MoveL RelTool (p1,32.000000,16.000000,15.618348,\Rx:=0.000000,\Ry:=-3.162780),vel1,zoneval,Extruder\WObj:=Workobject_1;
MoveL RelTool (p1,34.500000,16.000000,16.195789,\Rx:=0.000000,\Ry:=-2.451727),vel1,zoneval,Extruder\WObj:=Workobject_1;
MoveL RelTool (p1,37.000000,16.000000,16.604171,\Rx:=0.000000,\Ry:=-1.580071),vel1,zoneval,Extruder\WObj:=Workobject_1;
MoveL RelTool (p1,39.500000,16.000000,16.864821,\Rx:=0.000000,\Ry:=-1.023091),vel1,zoneval,Extruder\WObj:=Workobject_1;
MoveL RelTool (p1,42.000000,16.000000,16.985827,\Rx:=0.000000,\Ry:=-0.098788),vel1,zoneval,Extruder\WObj:=Workobject_1;
MoveL RelTool (p1,44.500000,16.000000,16.964311,\Rx:=0.000000,\Ry:=0.392042),vel1,zoneval,Extruder\WObj:=Workobject_1;
MoveL RelTool (p1,47.000000,16.000000,16.814464,\Rx:=0.000000,\Ry:=1.375711),vel1,zoneval,Extruder\WObj:=Workobject_1;
MoveL RelTool (p1,49.500000,16.000000,16.508665,\Rx:=0.000000,\Ry:=1.876566),vel1,zoneval,Extruder\WObj:=Workobject_1;
MoveL RelTool (p1,52.000000,16.000000,16.062619,\Rx:=0.000000,\Ry:=2.914714),vel1,zoneval,Extruder\WObj:=Workobject_1;
MoveL RelTool (p1,54.500000,16.000000,15.430893,\Rx:=0.000000,\Ry:=3.587334),vel1,zoneval,Extruder\WObj:=Workobject_1;
MoveL RelTool (p1,57.000000,16.000000,14.596569,\Rx:=0.000000,\Ry:=4.605885),vel1,zoneval,Extruder\WObj:=Workobject_1;
MoveL RelTool (p1,59.500000,16.000000,13.508587,\Rx:=0.000000,\Ry:=5.885518),vel1,zoneval,Extruder\WObj:=Workobject_1;
MoveL RelTool (p1,62.000000,16.000000,12.049469,\Rx:=0.000000,\Ry:=8.052866),vel1,zoneval,Extruder\WObj:=Workobject_1;
MoveL RelTool (p1,64.500000,16.000000,9.870531,\Rx:=0.000000,\Ry:=11.251023),vel1,zoneval,Extruder\WObj:=Workobject_1;
MoveL RelTool (p1,67.000000,16.000000,7.452288,\Rx:=0.000000,\Ry:=5.136110),vel1,zoneval,Extruder\WObj:=Workobject_1;
MoveL RelTool (p1,69.500000,16.000000,7.000000,\Rx:=0.000000,\Ry:=-0.000000),vel1,zoneval,Extruder\WObj:=Workobject_1;
MoveL RelTool (p1,72.000000,16.000000,7.000000,\Rx:=0.000000,\Ry:=-0.000000),vel1,zoneval,Extruder\WObj:=Workobject_1;
MoveL RelTool (p1,74.500000,16.000000,7.000000,\Rx:=0.000000,\Ry:=-0.000000),vel1,zoneval,Extruder\WObj:=Workobject_1;
MoveL RelTool (p1,77.000000,16.000000,7.000000,\Rx:=0.000000,\Ry:=-0.000000),vel1,zoneval,Extruder\WObj:=Workobject_1;
MoveL RelTool (p1,79.500000,16.000000,7.000000,\Rx:=0.000000,\Ry:=-0.000000),vel1,zoneval,Extruder\WObj:=Workobject_1;
MoveL RelTool (p1,82.000000,16.000000,7.000000,\Rx:=0.000000,\Ry:=-0.000000),vel1,zoneval,Extruder\WObj:=Workobject_1;




MoveL RelTool (p1,82.000000,16.000000,70.000000,\Rx:=0.000000,\Ry:=-0.000000),vel1,zoneval,Extruder\WObj:=Workobject_1;


MoveL RelTool (p1,3.000000,3.000000,70.00000,\Rx:=0.000000,\Ry:=0.000000),vel1,z0,Extruder\WObj:=Workobject_1;


MoveL RelTool (p1,3.000000,3.000000,7.500000,\Rx:=0.000000,\Ry:=0.000000),vel1,z0,Extruder\WObj:=Workobject_1;
MoveL RelTool (p1,16.889791,3.000000,7.500000,\Rx:=0.000000,\Ry:=0.000000),vel1,z0,Extruder\WObj:=Workobject_1;
MoveL RelTool (p1,17.532421,3.000000,7.551959,\Rx:=0.000000,\Ry:=0.000000),vel1,z0,Extruder\WObj:=Workobject_1;
MoveL RelTool (p1,18.158356,3.000000,7.706487,\Rx:=0.000000,\Ry:=0.000000),vel1,z0,Extruder\WObj:=Workobject_1;
MoveL RelTool (p1,18.751335,3.000000,7.959569,\Rx:=0.000000,\Ry:=0.000000),vel1,z0,Extruder\WObj:=Workobject_1;
MoveL RelTool (p1,19.295952,3.000000,8.304629,\Rx:=0.000000,\Ry:=0.000000),vel1,z0,Extruder\WObj:=Workobject_1;
MoveL RelTool (p1,19.778055,3.000000,8.732704,\Rx:=0.000000,\Ry:=0.000000),vel1,z0,Extruder\WObj:=Workobject_1;
MoveL RelTool (p1,20.185125,3.000000,9.232673,\Rx:=0.000000,\Ry:=0.000000),vel1,z0,Extruder\WObj:=Workobject_1;
MoveL RelTool (p1,20.434406,3.000000,9.577575,\Rx:=0.000000,\Ry:=0.000000),vel1,z0,Extruder\WObj:=Workobject_1;
MoveL RelTool (p1,21.354332,3.000000,10.637746,\Rx:=0.000000,\Ry:=0.000000),vel1,z0,Extruder\WObj:=Workobject_1;
MoveL RelTool (p1,22.624866,3.000000,11.778059,\Rx:=0.000000,\Ry:=0.000000),vel1,z0,Extruder\WObj:=Workobject_1;
MoveL RelTool (p1,24.188330,3.000000,12.885570,\Rx:=0.000000,\Ry:=0.000000),vel1,z0,Extruder\WObj:=Workobject_1;
MoveL RelTool (p1,26.083382,3.000000,13.951722,\Rx:=0.000000,\Ry:=0.000000),vel1,z0,Extruder\WObj:=Workobject_1;
MoveL RelTool (p1,28.279192,3.000000,14.927603,\Rx:=0.000000,\Ry:=0.000000),vel1,z0,Extruder\WObj:=Workobject_1;
MoveL RelTool (p1,30.704315,3.000000,15.771751,\Rx:=0.000000,\Ry:=0.000000),vel1,z0,Extruder\WObj:=Workobject_1;
MoveL RelTool (p1,33.363621,3.000000,16.473523,\Rx:=0.000000,\Ry:=0.000000),vel1,z0,Extruder\WObj:=Workobject_1;
MoveL RelTool (p1,36.232094,3.000000,17.007633,\Rx:=0.000000,\Ry:=0.000000),vel1,z0,Extruder\WObj:=Workobject_1;
MoveL RelTool (p1,39.211102,3.000000,17.350134,\Rx:=0.000000,\Ry:=0.000000),vel1,z0,Extruder\WObj:=Workobject_1;
MoveL RelTool (p1,42.244740,3.000000,17.495073,\Rx:=0.000000,\Ry:=0.000000),vel1,z0,Extruder\WObj:=Workobject_1;
MoveL RelTool (p1,45.290798,3.000000,17.438496,\Rx:=0.000000,\Ry:=0.000000),vel1,z0,Extruder\WObj:=Workobject_1;
MoveL RelTool (p1,48.269035,3.000000,17.185968,\Rx:=0.000000,\Ry:=0.000000),vel1,z0,Extruder\WObj:=Workobject_1;
MoveL RelTool (p1,51.111694,3.000000,16.752958,\Rx:=0.000000,\Ry:=0.000000),vel1,z0,Extruder\WObj:=Workobject_1;
MoveL RelTool (p1,53.811565,3.000000,16.146063,\Rx:=0.000000,\Ry:=0.000000),vel1,z0,Extruder\WObj:=Workobject_1;
MoveL RelTool (p1,56.313255,3.000000,15.385991,\Rx:=0.000000,\Ry:=0.000000),vel1,z0,Extruder\WObj:=Workobject_1;
MoveL RelTool (p1,58.536770,3.000000,14.519064,\Rx:=0.000000,\Ry:=0.000000),vel1,z0,Extruder\WObj:=Workobject_1;
MoveL RelTool (p1,60.496769,3.000000,13.560389,\Rx:=0.000000,\Ry:=0.000000),vel1,z0,Extruder\WObj:=Workobject_1;
MoveL RelTool (p1,62.188400,3.000000,12.528250,\Rx:=0.000000,\Ry:=0.000000),vel1,z0,Extruder\WObj:=Workobject_1;
MoveL RelTool (p1,63.608570,3.000000,11.447268,\Rx:=0.000000,\Ry:=0.000000),vel1,z0,Extruder\WObj:=Workobject_1;
MoveL RelTool (p1,64.754211,3.000000,10.346784,\Rx:=0.000000,\Ry:=0.000000),vel1,z0,Extruder\WObj:=Workobject_1;
MoveL RelTool (p1,65.647247,3.000000,9.232673,\Rx:=0.000000,\Ry:=0.000000),vel1,z0,Extruder\WObj:=Workobject_1;
MoveL RelTool (p1,66.054314,3.000000,8.732704,\Rx:=0.000000,\Ry:=0.000000),vel1,z0,Extruder\WObj:=Workobject_1;
MoveL RelTool (p1,66.536423,3.000000,8.304629,\Rx:=0.000000,\Ry:=0.000000),vel1,z0,Extruder\WObj:=Workobject_1;
MoveL RelTool (p1,67.081032,3.000000,7.959569,\Rx:=0.000000,\Ry:=0.000000),vel1,z0,Extruder\WObj:=Workobject_1;
MoveL RelTool (p1,67.674019,3.000000,7.706487,\Rx:=0.000000,\Ry:=0.000000),vel1,z0,Extruder\WObj:=Workobject_1;
MoveL RelTool (p1,68.299950,3.000000,7.551959,\Rx:=0.000000,\Ry:=0.000000),vel1,z0,Extruder\WObj:=Workobject_1;
MoveL RelTool (p1,68.942581,3.000000,7.500000,\Rx:=0.000000,\Ry:=0.000000),vel1,z0,Extruder\WObj:=Workobject_1;
MoveL RelTool (p1,82.832375,3.000000,7.500000,\Rx:=0.000000,\Ry:=0.000000),vel1,z0,Extruder\WObj:=Workobject_1;
MoveL RelTool (p1,82.832375,16.000000,7.500000,\Rx:=0.000000,\Ry:=0.000000),vel1,z0,Extruder\WObj:=Workobject_1;
MoveL RelTool (p1,68.942581,16.000000,7.500000,\Rx:=0.000000,\Ry:=0.000000),vel1,z0,Extruder\WObj:=Workobject_1;
MoveL RelTool (p1,68.299950,16.000000,7.551959,\Rx:=0.000000,\Ry:=0.000000),vel1,z0,Extruder\WObj:=Workobject_1;
MoveL RelTool (p1,67.674019,16.000000,7.706487,\Rx:=0.000000,\Ry:=0.000000),vel1,z0,Extruder\WObj:=Workobject_1;
MoveL RelTool (p1,67.081032,16.000000,7.959569,\Rx:=0.000000,\Ry:=0.000000),vel1,z0,Extruder\WObj:=Workobject_1;
MoveL RelTool (p1,66.536423,16.000000,8.304629,\Rx:=0.000000,\Ry:=0.000000),vel1,z0,Extruder\WObj:=Workobject_1;
MoveL RelTool (p1,66.054314,16.000000,8.732704,\Rx:=0.000000,\Ry:=0.000000),vel1,z0,Extruder\WObj:=Workobject_1;
MoveL RelTool (p1,65.647247,16.000000,9.232673,\Rx:=0.000000,\Ry:=0.000000),vel1,z0,Extruder\WObj:=Workobject_1;
MoveL RelTool (p1,65.163933,16.000000,9.874841,\Rx:=0.000000,\Ry:=0.000000),vel1,z0,Extruder\WObj:=Workobject_1;
MoveL RelTool (p1,64.749672,16.000000,10.342769,\Rx:=0.000000,\Ry:=0.000000),vel1,z0,Extruder\WObj:=Workobject_1;
MoveL RelTool (p1,64.601288,16.000000,10.510382,\Rx:=0.000000,\Ry:=0.000000),vel1,z0,Extruder\WObj:=Workobject_1;
MoveL RelTool (p1,63.937405,16.000000,11.157751,\Rx:=0.000000,\Ry:=0.000000),vel1,z0,Extruder\WObj:=Workobject_1;
MoveL RelTool (p1,63.603333,16.000000,11.441092,\Rx:=0.000000,\Ry:=0.000000),vel1,z0,Extruder\WObj:=Workobject_1;
MoveL RelTool (p1,63.179665,16.000000,11.800433,\Rx:=0.000000,\Ry:=0.000000),vel1,z0,Extruder\WObj:=Workobject_1;
MoveL RelTool (p1,62.342442,16.000000,12.422123,\Rx:=0.000000,\Ry:=0.000000),vel1,z0,Extruder\WObj:=Workobject_1;
MoveL RelTool (p1,62.185829,16.000000,12.524306,\Rx:=0.000000,\Ry:=0.000000),vel1,z0,Extruder\WObj:=Workobject_1;
MoveL RelTool (p1,61.383541,16.000000,13.047758,\Rx:=0.000000,\Ry:=0.000000),vel1,z0,Extruder\WObj:=Workobject_1;
MoveL RelTool (p1,60.495010,16.000000,13.557323,\Rx:=0.000000,\Ry:=0.000000),vel1,z0,Extruder\WObj:=Workobject_1;
MoveL RelTool (p1,60.358730,16.000000,13.635481,\Rx:=0.000000,\Ry:=0.000000),vel1,z0,Extruder\WObj:=Workobject_1;
MoveL RelTool (p1,59.242863,16.000000,14.198255,\Rx:=0.000000,\Ry:=0.000000),vel1,z0,Extruder\WObj:=Workobject_1;
MoveL RelTool (p1,58.533695,16.000000,14.512110,\Rx:=0.000000,\Ry:=0.000000),vel1,z0,Extruder\WObj:=Workobject_1;
MoveL RelTool (p1,58.030029,16.000000,14.735016,\Rx:=0.000000,\Ry:=0.000000),vel1,z0,Extruder\WObj:=Workobject_1;
MoveL RelTool (p1,56.707867,16.000000,15.246546,\Rx:=0.000000,\Ry:=0.000000),vel1,z0,Extruder\WObj:=Workobject_1;
MoveL RelTool (p1,56.311142,16.000000,15.379692,\Rx:=0.000000,\Ry:=0.000000),vel1,z0,Extruder\WObj:=Workobject_1;
MoveL RelTool (p1,55.286888,16.000000,15.723446,\Rx:=0.000000,\Ry:=0.000000),vel1,z0,Extruder\WObj:=Workobject_1;
MoveL RelTool (p1,53.819916,16.000000,16.144513,\Rx:=0.000000,\Ry:=0.000000),vel1,z0,Extruder\WObj:=Workobject_1;
MoveL RelTool (p1,53.811668,16.000000,16.146502,\Rx:=0.000000,\Ry:=0.000000),vel1,z0,Extruder\WObj:=Workobject_1;
MoveL RelTool (p1,52.291843,16.000000,16.513170,\Rx:=0.000000,\Ry:=0.000000),vel1,z0,Extruder\WObj:=Workobject_1;
MoveL RelTool (p1,51.110493,16.000000,16.746876,\Rx:=0.000000,\Ry:=0.000000),vel1,z0,Extruder\WObj:=Workobject_1;
MoveL RelTool (p1,50.699913,16.000000,16.828100,\Rx:=0.000000,\Ry:=0.000000),vel1,z0,Extruder\WObj:=Workobject_1;
MoveL RelTool (p1,49.040199,16.000000,17.087831,\Rx:=0.000000,\Ry:=0.000000),vel1,z0,Extruder\WObj:=Workobject_1;
MoveL RelTool (p1,48.268082,16.000000,17.177822,\Rx:=0.000000,\Ry:=0.000000),vel1,z0,Extruder\WObj:=Workobject_1;
MoveL RelTool (p1,47.334873,16.000000,17.286589,\Rx:=0.000000,\Ry:=0.000000),vel1,z0,Extruder\WObj:=Workobject_1;
MoveL RelTool (p1,45.589977,16.000000,17.422077,\Rx:=0.000000,\Ry:=0.000000),vel1,z0,Extruder\WObj:=Workobject_1;
MoveL RelTool (p1,45.290615,16.000000,17.433790,\Rx:=0.000000,\Ry:=0.000000),vel1,z0,Extruder\WObj:=Workobject_1;
MoveL RelTool (p1,43.831112,16.000000,17.490894,\Rx:=0.000000,\Ry:=0.000000),vel1,z0,Extruder\WObj:=Workobject_1;
MoveL RelTool (p1,42.244736,16.000000,17.492092,\Rx:=0.000000,\Ry:=0.000000),vel1,z0,Extruder\WObj:=Workobject_1;
MoveL RelTool (p1,42.070164,16.000000,17.492224,\Rx:=0.000000,\Ry:=0.000000),vel1,z0,Extruder\WObj:=Workobject_1;
MoveL RelTool (p1,40.311550,16.000000,17.426056,\Rx:=0.000000,\Ry:=0.000000),vel1,z0,Extruder\WObj:=Workobject_1;
MoveL RelTool (p1,39.211697,16.000000,17.342295,\Rx:=0.000000,\Ry:=0.000000),vel1,z0,Extruder\WObj:=Workobject_1;
MoveL RelTool (p1,38.562359,16.000000,17.292841,\Rx:=0.000000,\Ry:=0.000000),vel1,z0,Extruder\WObj:=Workobject_1;
MoveL RelTool (p1,36.841461,16.000000,17.094522,\Rx:=0.000000,\Ry:=0.000000),vel1,z0,Extruder\WObj:=Workobject_1;
MoveL RelTool (p1,36.233295,16.000000,16.999901,\Rx:=0.000000,\Ry:=0.000000),vel1,z0,Extruder\WObj:=Workobject_1;
MoveL RelTool (p1,35.157150,16.000000,16.832468,\Rx:=0.000000,\Ry:=0.000000),vel1,z0,Extruder\WObj:=Workobject_1;
MoveL RelTool (p1,33.534817,16.000000,16.511932,\Rx:=0.000000,\Ry:=0.000000),vel1,z0,Extruder\WObj:=Workobject_1;
MoveL RelTool (p1,33.364307,16.000000,16.470687,\Rx:=0.000000,\Ry:=0.000000),vel1,z0,Extruder\WObj:=Workobject_1;
MoveL RelTool (p1,31.975235,16.000000,16.134667,\Rx:=0.000000,\Ry:=0.000000),vel1,z0,Extruder\WObj:=Workobject_1;
MoveL RelTool (p1,30.705374,16.000000,15.768086,\Rx:=0.000000,\Ry:=0.000000),vel1,z0,Extruder\WObj:=Workobject_1;
MoveL RelTool (p1,30.481377,16.000000,15.703423,\Rx:=0.000000,\Ry:=0.000000),vel1,z0,Extruder\WObj:=Workobject_1;
MoveL RelTool (p1,29.050327,16.000000,15.219646,\Rx:=0.000000,\Ry:=0.000000),vel1,z0,Extruder\WObj:=Workobject_1;
MoveL RelTool (p1,28.282177,16.000000,14.919954,\Rx:=0.000000,\Ry:=0.000000),vel1,z0,Extruder\WObj:=Workobject_1;
MoveL RelTool (p1,27.714354,16.000000,14.698419,\Rx:=0.000000,\Ry:=0.000000),vel1,z0,Extruder\WObj:=Workobject_1;
MoveL RelTool (p1,26.464403,16.000000,14.138699,\Rx:=0.000000,\Ry:=0.000000),vel1,z0,Extruder\WObj:=Workobject_1;
MoveL RelTool (p1,26.086796,16.000000,13.945067,\Rx:=0.000000,\Ry:=0.000000),vel1,z0,Extruder\WObj:=Workobject_1;
MoveL RelTool (p1,25.315779,16.000000,13.549702,\Rx:=0.000000,\Ry:=0.000000),vel1,z0,Extruder\WObj:=Workobject_1;
MoveL RelTool (p1,24.267054,16.000000,12.935243,\Rx:=0.000000,\Ry:=0.000000),vel1,z0,Extruder\WObj:=Workobject_1;
MoveL RelTool (p1,24.189692,16.000000,12.883533,\Rx:=0.000000,\Ry:=0.000000),vel1,z0,Extruder\WObj:=Workobject_1;
MoveL RelTool (p1,23.318321,16.000000,12.301085,\Rx:=0.000000,\Ry:=0.000000),vel1,z0,Extruder\WObj:=Workobject_1;
MoveL RelTool (p1,22.627743,16.000000,11.774289,\Rx:=0.000000,\Ry:=0.000000),vel1,z0,Extruder\WObj:=Workobject_1;
MoveL RelTool (p1,22.482136,16.000000,11.663216,\Rx:=0.000000,\Ry:=0.000000),vel1,z0,Extruder\WObj:=Workobject_1;
MoveL RelTool (p1,21.725685,16.000000,11.001189,\Rx:=0.000000,\Ry:=0.000000),vel1,z0,Extruder\WObj:=Workobject_1;
MoveL RelTool (p1,21.360172,16.000000,10.631966,\Rx:=0.000000,\Ry:=0.000000),vel1,z0,Extruder\WObj:=Workobject_1;
MoveL RelTool (p1,21.079424,16.000000,10.348370,\Rx:=0.000000,\Ry:=0.000000),vel1,z0,Extruder\WObj:=Workobject_1;
MoveL RelTool (p1,20.517708,16.000000,9.686148,\Rx:=0.000000,\Ry:=0.000000),vel1,z0,Extruder\WObj:=Workobject_1;
MoveL RelTool (p1,20.436796,16.000000,9.575823,\Rx:=0.000000,\Ry:=0.000000),vel1,z0,Extruder\WObj:=Workobject_1;
MoveL RelTool (p1,20.185125,16.000000,9.232673,\Rx:=0.000000,\Ry:=0.000000),vel1,z0,Extruder\WObj:=Workobject_1;
MoveL RelTool (p1,19.778055,16.000000,8.732704,\Rx:=0.000000,\Ry:=0.000000),vel1,z0,Extruder\WObj:=Workobject_1;
MoveL RelTool (p1,19.295952,16.000000,8.304629,\Rx:=0.000000,\Ry:=0.000000),vel1,z0,Extruder\WObj:=Workobject_1;
MoveL RelTool (p1,18.751335,16.000000,7.959569,\Rx:=0.000000,\Ry:=0.000000),vel1,z0,Extruder\WObj:=Workobject_1;
MoveL RelTool (p1,18.158356,16.000000,7.706487,\Rx:=0.000000,\Ry:=0.000000),vel1,z0,Extruder\WObj:=Workobject_1;
MoveL RelTool (p1,17.532421,16.000000,7.551959,\Rx:=0.000000,\Ry:=0.000000),vel1,z0,Extruder\WObj:=Workobject_1;
MoveL RelTool (p1,16.889791,16.000000,7.500000,\Rx:=0.000000,\Ry:=0.000000),vel1,z0,Extruder\WObj:=Workobject_1;
MoveL RelTool (p1,3.000000,16.000000,7.500000,\Rx:=0.000000,\Ry:=0.000000),vel1,z0,Extruder\WObj:=Workobject_1;
MoveL RelTool (p1,3.000000,3.000000,7.500000,\Rx:=0.000000,\Ry:=0.000000),vel1,z0,Extruder\WObj:=Workobject_1;



MoveL RelTool (p1,3.000000,3.000000,7.500000,\Rx:=0.000000,\Ry:=0),vel1,zoneval,Extruder\WObj:=Workobject_1;
MoveL RelTool (p1,5.000000,3.000000,7.500000,\Rx:=0.000000,\Ry:=-0.000000),vel1,zoneval,Extruder\WObj:=Workobject_1;
MoveL RelTool (p1,7.500000,3.000000,7.500000,\Rx:=0.000000,\Ry:=-0.000000),vel1,zoneval,Extruder\WObj:=Workobject_1;
MoveL RelTool (p1,10.000000,3.000000,7.500000,\Rx:=0.000000,\Ry:=-0.000000),vel1,zoneval,Extruder\WObj:=Workobject_1;
MoveL RelTool (p1,12.500000,3.000000,7.500000,\Rx:=0.000000,\Ry:=-0.000000),vel1,zoneval,Extruder\WObj:=Workobject_1;
MoveL RelTool (p1,15.000000,3.000000,7.500000,\Rx:=0.000000,\Ry:=-0.000000),vel1,zoneval,Extruder\WObj:=Workobject_1;
MoveL RelTool (p1,17.500000,3.000000,7.549338,\Rx:=0.000000,\Ry:=-2.952187),vel1,zoneval,Extruder\WObj:=Workobject_1;
MoveL RelTool (p1,20.000000,3.000000,9.005299,\Rx:=0.000000,\Ry:=-11.631209),vel1,zoneval,Extruder\WObj:=Workobject_1;
MoveL RelTool (p1,22.500000,3.000000,11.665991,\Rx:=0.000000,\Ry:=-8.238851),vel1,zoneval,Extruder\WObj:=Workobject_1;
MoveL RelTool (p1,25.000000,3.000000,13.342214,\Rx:=0.000000,\Ry:=-6.524894),vel1,zoneval,Extruder\WObj:=Workobject_1;
MoveL RelTool (p1,27.500000,3.000000,14.581308,\Rx:=0.000000,\Ry:=-5.324828),vel1,zoneval,Extruder\WObj:=Workobject_1;
MoveL RelTool (p1,30.000000,3.000000,15.526590,\Rx:=0.000000,\Ry:=-4.264941),vel1,zoneval,Extruder\WObj:=Workobject_1;
MoveL RelTool (p1,32.500000,3.000000,16.245620,\Rx:=0.000000,\Ry:=-3.285097),vel1,zoneval,Extruder\WObj:=Workobject_1;
MoveL RelTool (p1,35.000000,3.000000,16.778217,\Rx:=0.000000,\Ry:=-2.343931),vel1,zoneval,Extruder\WObj:=Workobject_1;
MoveL RelTool (p1,37.500000,3.000000,17.153406,\Rx:=0.000000,\Ry:=-1.457462),vel1,zoneval,Extruder\WObj:=Workobject_1;
MoveL RelTool (p1,40.000000,3.000000,17.387825,\Rx:=0.000000,\Ry:=-0.607859),vel1,zoneval,Extruder\WObj:=Workobject_1;
MoveL RelTool (p1,42.500000,3.000000,17.490332,\Rx:=0.000000,\Ry:=0.236465),vel1,zoneval,Extruder\WObj:=Workobject_1;
MoveL RelTool (p1,45.000000,3.000000,17.443897,\Rx:=0.000000,\Ry:=0.588828),vel1,zoneval,Extruder\WObj:=Workobject_1;
MoveL RelTool (p1,47.500000,3.000000,17.251176,\Rx:=0.000000,\Ry:=1.077014),vel1,zoneval,Extruder\WObj:=Workobject_1;
MoveL RelTool (p1,50.000000,3.000000,16.922298,\Rx:=0.000000,\Ry:=1.924676),vel1,zoneval,Extruder\WObj:=Workobject_1;
MoveL RelTool (p1,52.500000,3.000000,16.440885,\Rx:=0.000000,\Ry:=2.815279),vel1,zoneval,Extruder\WObj:=Workobject_1;
MoveL RelTool (p1,55.000000,3.000000,15.784989,\Rx:=0.000000,\Ry:=3.755557),vel1,zoneval,Extruder\WObj:=Workobject_1;
MoveL RelTool (p1,57.500000,3.000000,14.923291,\Rx:=0.000000,\Ry:=4.733408),vel1,zoneval,Extruder\WObj:=Workobject_1;
MoveL RelTool (p1,60.000000,3.000000,13.803368,\Rx:=0.000000,\Ry:=5.800076),vel1,zoneval,Extruder\WObj:=Workobject_1;
MoveL RelTool (p1,62.500000,3.000000,12.291071,\Rx:=0.000000,\Ry:=8.283792),vel1,zoneval,Extruder\WObj:=Workobject_1;
MoveL RelTool (p1,65.000000,3.000000,10.040149,\Rx:=0.000000,\Ry:=11.396766),vel1,zoneval,Extruder\WObj:=Workobject_1;
MoveL RelTool (p1,67.500000,3.000000,7.780757,\Rx:=0.000000,\Ry:=3.821551),vel1,zoneval,Extruder\WObj:=Workobject_1;
MoveL RelTool (p1,70.000000,3.000000,7.500000,\Rx:=0.000000,\Ry:=-0.000000),vel1,zoneval,Extruder\WObj:=Workobject_1;
MoveL RelTool (p1,72.500000,3.000000,7.500000,\Rx:=0.000000,\Ry:=-0.000000),vel1,zoneval,Extruder\WObj:=Workobject_1;
MoveL RelTool (p1,75.000000,3.000000,7.500000,\Rx:=0.000000,\Ry:=-0.000000),vel1,zoneval,Extruder\WObj:=Workobject_1;
MoveL RelTool (p1,77.500000,3.000000,7.500000,\Rx:=0.000000,\Ry:=-0.000000),vel1,zoneval,Extruder\WObj:=Workobject_1;
MoveL RelTool (p1,80.000000,3.000000,7.500000,\Rx:=0.000000,\Ry:=-0.000000),vel1,zoneval,Extruder\WObj:=Workobject_1;
MoveL RelTool (p1,82.500000,3.000000,7.500000,\Rx:=0.000000,\Ry:=-0.000000),vel1,zoneval,Extruder\WObj:=Workobject_1;
MoveL RelTool (p1,80.500000,3.500000,7.500000,\Rx:=0.000000,\Ry:=0.000000),vel1,zoneval,Extruder\WObj:=Workobject_1;
MoveL RelTool (p1,78.000000,3.500000,7.500000,\Rx:=0.000000,\Ry:=0.000000),vel1,zoneval,Extruder\WObj:=Workobject_1;
MoveL RelTool (p1,75.500000,3.500000,7.500000,\Rx:=0.000000,\Ry:=0.000000),vel1,zoneval,Extruder\WObj:=Workobject_1;
MoveL RelTool (p1,73.000000,3.500000,7.500000,\Rx:=0.000000,\Ry:=0.000000),vel1,zoneval,Extruder\WObj:=Workobject_1;
MoveL RelTool (p1,70.500000,3.500000,7.500000,\Rx:=0.000000,\Ry:=0.000000),vel1,zoneval,Extruder\WObj:=Workobject_1;
MoveL RelTool (p1,68.000000,3.500000,7.626010,\Rx:=0.000000,\Ry:=3.821551),vel1,zoneval,Extruder\WObj:=Workobject_1;
MoveL RelTool (p1,65.500000,3.500000,9.417880,\Rx:=0.000000,\Ry:=11.396766),vel1,zoneval,Extruder\WObj:=Workobject_1;
MoveL RelTool (p1,63.000000,3.500000,11.911517,\Rx:=0.000000,\Ry:=8.283792),vel1,zoneval,Extruder\WObj:=Workobject_1;
MoveL RelTool (p1,60.500000,3.500000,13.558379,\Rx:=0.000000,\Ry:=5.806843),vel1,zoneval,Extruder\WObj:=Workobject_1;
MoveL RelTool (p1,58.000000,3.500000,14.729052,\Rx:=0.000000,\Ry:=4.733408),vel1,zoneval,Extruder\WObj:=Workobject_1;
MoveL RelTool (p1,55.500000,3.500000,15.633095,\Rx:=0.000000,\Ry:=3.755557),vel1,zoneval,Extruder\WObj:=Workobject_1;
MoveL RelTool (p1,53.000000,3.500000,16.329473,\Rx:=0.000000,\Ry:=2.815279),vel1,zoneval,Extruder\WObj:=Workobject_1;
MoveL RelTool (p1,50.500000,3.500000,16.846613,\Rx:=0.000000,\Ry:=1.924676),vel1,zoneval,Extruder\WObj:=Workobject_1;
MoveL RelTool (p1,48.000000,3.500000,17.209604,\Rx:=0.000000,\Ry:=1.077014),vel1,zoneval,Extruder\WObj:=Workobject_1;
MoveL RelTool (p1,45.500000,3.500000,17.421581,\Rx:=0.000000,\Ry:=0.592614),vel1,zoneval,Extruder\WObj:=Workobject_1;
MoveL RelTool (p1,43.000000,3.500000,17.482018,\Rx:=0.000000,\Ry:=0.236465),vel1,zoneval,Extruder\WObj:=Workobject_1;
MoveL RelTool (p1,40.500000,3.500000,17.412612,\Rx:=0.000000,\Ry:=-0.607859),vel1,zoneval,Extruder\WObj:=Workobject_1;
MoveL RelTool (p1,38.000000,3.500000,17.211557,\Rx:=0.000000,\Ry:=-1.457462),vel1,zoneval,Extruder\WObj:=Workobject_1;
MoveL RelTool (p1,35.500000,3.500000,16.871568,\Rx:=0.000000,\Ry:=-2.343931),vel1,zoneval,Extruder\WObj:=Workobject_1;
MoveL RelTool (p1,33.000000,3.500000,16.378625,\Rx:=0.000000,\Ry:=-3.285097),vel1,zoneval,Extruder\WObj:=Workobject_1;
MoveL RelTool (p1,30.500000,3.500000,15.700989,\Rx:=0.000000,\Ry:=-4.264941),vel1,zoneval,Extruder\WObj:=Workobject_1;
MoveL RelTool (p1,28.000000,3.500000,14.804200,\Rx:=0.000000,\Ry:=-5.324828),vel1,zoneval,Extruder\WObj:=Workobject_1;
MoveL RelTool (p1,25.500000,3.500000,13.624660,\Rx:=0.000000,\Ry:=-6.524894),vel1,zoneval,Extruder\WObj:=Workobject_1;
MoveL RelTool (p1,23.000000,3.500000,12.045016,\Rx:=0.000000,\Ry:=-8.250405),vel1,zoneval,Extruder\WObj:=Workobject_1;
MoveL RelTool (p1,20.500000,3.500000,9.654224,\Rx:=0.000000,\Ry:=-11.641231),vel1,zoneval,Extruder\WObj:=Workobject_1;
MoveL RelTool (p1,18.000000,3.500000,7.667393,\Rx:=0.000000,\Ry:=-2.952187),vel1,zoneval,Extruder\WObj:=Workobject_1;
MoveL RelTool (p1,15.500000,3.500000,7.500000,\Rx:=0.000000,\Ry:=0.000000),vel1,zoneval,Extruder\WObj:=Workobject_1;
MoveL RelTool (p1,13.000000,3.500000,7.500000,\Rx:=0.000000,\Ry:=0.000000),vel1,zoneval,Extruder\WObj:=Workobject_1;
MoveL RelTool (p1,10.500000,3.500000,7.500000,\Rx:=0.000000,\Ry:=0.000000),vel1,zoneval,Extruder\WObj:=Workobject_1;
MoveL RelTool (p1,8.000000,3.500000,7.500000,\Rx:=0.000000,\Ry:=0.000000),vel1,zoneval,Extruder\WObj:=Workobject_1;
MoveL RelTool (p1,5.500000,3.500000,7.500000,\Rx:=0.000000,\Ry:=0.000000),vel1,zoneval,Extruder\WObj:=Workobject_1;
MoveL RelTool (p1,3.000000,3.500000,7.500000,\Rx:=0.000000,\Ry:=0.000000),vel1,zoneval,Extruder\WObj:=Workobject_1;
MoveL RelTool (p1,5.000000,4.000000,7.500000,\Rx:=0.000000,\Ry:=-0.000000),vel1,zoneval,Extruder\WObj:=Workobject_1;
MoveL RelTool (p1,7.500000,4.000000,7.500000,\Rx:=0.000000,\Ry:=-0.000000),vel1,zoneval,Extruder\WObj:=Workobject_1;
MoveL RelTool (p1,10.000000,4.000000,7.500000,\Rx:=0.000000,\Ry:=-0.000000),vel1,zoneval,Extruder\WObj:=Workobject_1;
MoveL RelTool (p1,12.500000,4.000000,7.500000,\Rx:=0.000000,\Ry:=-0.000000),vel1,zoneval,Extruder\WObj:=Workobject_1;
MoveL RelTool (p1,15.000000,4.000000,7.500000,\Rx:=0.000000,\Ry:=-0.000000),vel1,zoneval,Extruder\WObj:=Workobject_1;
MoveL RelTool (p1,17.500000,4.000000,7.549338,\Rx:=0.000000,\Ry:=-2.952187),vel1,zoneval,Extruder\WObj:=Workobject_1;
MoveL RelTool (p1,20.000000,4.000000,9.005299,\Rx:=0.000000,\Ry:=-11.651234),vel1,zoneval,Extruder\WObj:=Workobject_1;
MoveL RelTool (p1,22.500000,4.000000,11.667010,\Rx:=0.000000,\Ry:=-8.261944),vel1,zoneval,Extruder\WObj:=Workobject_1;
MoveL RelTool (p1,25.000000,4.000000,13.344508,\Rx:=0.000000,\Ry:=-6.524894),vel1,zoneval,Extruder\WObj:=Workobject_1;
MoveL RelTool (p1,27.500000,4.000000,14.582665,\Rx:=0.000000,\Ry:=-5.324828),vel1,zoneval,Extruder\WObj:=Workobject_1;
MoveL RelTool (p1,30.000000,4.000000,15.527303,\Rx:=0.000000,\Ry:=-4.264941),vel1,zoneval,Extruder\WObj:=Workobject_1;
MoveL RelTool (p1,32.500000,4.000000,16.247737,\Rx:=0.000000,\Ry:=-3.285097),vel1,zoneval,Extruder\WObj:=Workobject_1;
MoveL RelTool (p1,35.000000,4.000000,16.778720,\Rx:=0.000000,\Ry:=-2.343931),vel1,zoneval,Extruder\WObj:=Workobject_1;
MoveL RelTool (p1,37.500000,4.000000,17.154736,\Rx:=0.000000,\Ry:=-1.457462),vel1,zoneval,Extruder\WObj:=Workobject_1;
MoveL RelTool (p1,40.000000,4.000000,17.389621,\Rx:=0.000000,\Ry:=-0.607859),vel1,zoneval,Extruder\WObj:=Workobject_1;
MoveL RelTool (p1,42.500000,4.000000,17.492277,\Rx:=0.000000,\Ry:=0.236465),vel1,zoneval,Extruder\WObj:=Workobject_1;
MoveL RelTool (p1,45.000000,4.000000,17.445842,\Rx:=0.000000,\Ry:=0.596401),vel1,zoneval,Extruder\WObj:=Workobject_1;
MoveL RelTool (p1,47.500000,4.000000,17.252823,\Rx:=0.000000,\Ry:=1.077014),vel1,zoneval,Extruder\WObj:=Workobject_1;
MoveL RelTool (p1,50.000000,4.000000,16.923253,\Rx:=0.000000,\Ry:=1.924676),vel1,zoneval,Extruder\WObj:=Workobject_1;
MoveL RelTool (p1,52.500000,4.000000,16.442847,\Rx:=0.000000,\Ry:=2.815279),vel1,zoneval,Extruder\WObj:=Workobject_1;
MoveL RelTool (p1,55.000000,4.000000,15.785025,\Rx:=0.000000,\Ry:=3.755557),vel1,zoneval,Extruder\WObj:=Workobject_1;
MoveL RelTool (p1,57.500000,4.000000,14.924704,\Rx:=0.000000,\Ry:=4.733408),vel1,zoneval,Extruder\WObj:=Workobject_1;
MoveL RelTool (p1,60.000000,4.000000,13.803951,\Rx:=0.000000,\Ry:=5.816036),vel1,zoneval,Extruder\WObj:=Workobject_1;
MoveL RelTool (p1,62.500000,4.000000,12.293125,\Rx:=0.000000,\Ry:=8.283792),vel1,zoneval,Extruder\WObj:=Workobject_1;
MoveL RelTool (p1,65.000000,4.000000,10.043165,\Rx:=0.000000,\Ry:=11.396766),vel1,zoneval,Extruder\WObj:=Workobject_1;
MoveL RelTool (p1,67.500000,4.000000,7.780757,\Rx:=0.000000,\Ry:=3.821551),vel1,zoneval,Extruder\WObj:=Workobject_1;
MoveL RelTool (p1,70.000000,4.000000,7.500000,\Rx:=0.000000,\Ry:=-0.000000),vel1,zoneval,Extruder\WObj:=Workobject_1;
MoveL RelTool (p1,72.500000,4.000000,7.500000,\Rx:=0.000000,\Ry:=-0.000000),vel1,zoneval,Extruder\WObj:=Workobject_1;
MoveL RelTool (p1,75.000000,4.000000,7.500000,\Rx:=0.000000,\Ry:=-0.000000),vel1,zoneval,Extruder\WObj:=Workobject_1;
MoveL RelTool (p1,77.500000,4.000000,7.500000,\Rx:=0.000000,\Ry:=-0.000000),vel1,zoneval,Extruder\WObj:=Workobject_1;
MoveL RelTool (p1,80.000000,4.000000,7.500000,\Rx:=0.000000,\Ry:=-0.000000),vel1,zoneval,Extruder\WObj:=Workobject_1;
MoveL RelTool (p1,82.500000,4.000000,7.500000,\Rx:=0.000000,\Ry:=-0.000000),vel1,zoneval,Extruder\WObj:=Workobject_1;
MoveL RelTool (p1,80.500000,4.500000,7.500000,\Rx:=0.000000,\Ry:=0.000000),vel1,zoneval,Extruder\WObj:=Workobject_1;
MoveL RelTool (p1,78.000000,4.500000,7.500000,\Rx:=0.000000,\Ry:=0.000000),vel1,zoneval,Extruder\WObj:=Workobject_1;
MoveL RelTool (p1,75.500000,4.500000,7.500000,\Rx:=0.000000,\Ry:=0.000000),vel1,zoneval,Extruder\WObj:=Workobject_1;
MoveL RelTool (p1,73.000000,4.500000,7.500000,\Rx:=0.000000,\Ry:=0.000000),vel1,zoneval,Extruder\WObj:=Workobject_1;
MoveL RelTool (p1,70.500000,4.500000,7.500000,\Rx:=0.000000,\Ry:=0.000000),vel1,zoneval,Extruder\WObj:=Workobject_1;
MoveL RelTool (p1,68.000000,4.500000,7.626010,\Rx:=0.000000,\Ry:=3.821551),vel1,zoneval,Extruder\WObj:=Workobject_1;
MoveL RelTool (p1,65.500000,4.500000,9.420896,\Rx:=0.000000,\Ry:=11.396766),vel1,zoneval,Extruder\WObj:=Workobject_1;
MoveL RelTool (p1,63.000000,4.500000,11.913570,\Rx:=0.000000,\Ry:=8.283792),vel1,zoneval,Extruder\WObj:=Workobject_1;
MoveL RelTool (p1,60.500000,4.500000,13.558066,\Rx:=0.000000,\Ry:=5.825222),vel1,zoneval,Extruder\WObj:=Workobject_1;
MoveL RelTool (p1,58.000000,4.500000,14.730466,\Rx:=0.000000,\Ry:=4.733408),vel1,zoneval,Extruder\WObj:=Workobject_1;
MoveL RelTool (p1,55.500000,4.500000,15.633131,\Rx:=0.000000,\Ry:=3.755557),vel1,zoneval,Extruder\WObj:=Workobject_1;
MoveL RelTool (p1,53.000000,4.500000,16.331434,\Rx:=0.000000,\Ry:=2.815279),vel1,zoneval,Extruder\WObj:=Workobject_1;
MoveL RelTool (p1,50.500000,4.500000,16.847568,\Rx:=0.000000,\Ry:=1.924676),vel1,zoneval,Extruder\WObj:=Workobject_1;
MoveL RelTool (p1,48.000000,4.500000,17.211251,\Rx:=0.000000,\Ry:=1.077014),vel1,zoneval,Extruder\WObj:=Workobject_1;
MoveL RelTool (p1,45.500000,4.500000,17.423037,\Rx:=0.000000,\Ry:=0.605024),vel1,zoneval,Extruder\WObj:=Workobject_1;
MoveL RelTool (p1,43.000000,4.500000,17.483963,\Rx:=0.000000,\Ry:=0.236465),vel1,zoneval,Extruder\WObj:=Workobject_1;
MoveL RelTool (p1,40.500000,4.500000,17.414408,\Rx:=0.000000,\Ry:=-0.607859),vel1,zoneval,Extruder\WObj:=Workobject_1;
MoveL RelTool (p1,38.000000,4.500000,17.212887,\Rx:=0.000000,\Ry:=-1.457462),vel1,zoneval,Extruder\WObj:=Workobject_1;
MoveL RelTool (p1,35.500000,4.500000,16.872071,\Rx:=0.000000,\Ry:=-2.343931),vel1,zoneval,Extruder\WObj:=Workobject_1;
MoveL RelTool (p1,33.000000,4.500000,16.380743,\Rx:=0.000000,\Ry:=-3.285097),vel1,zoneval,Extruder\WObj:=Workobject_1;
MoveL RelTool (p1,30.500000,4.500000,15.701702,\Rx:=0.000000,\Ry:=-4.264941),vel1,zoneval,Extruder\WObj:=Workobject_1;
MoveL RelTool (p1,28.000000,4.500000,14.805557,\Rx:=0.000000,\Ry:=-5.324828),vel1,zoneval,Extruder\WObj:=Workobject_1;
MoveL RelTool (p1,25.500000,4.500000,13.626955,\Rx:=0.000000,\Ry:=-6.524894),vel1,zoneval,Extruder\WObj:=Workobject_1;
MoveL RelTool (p1,23.000000,4.500000,12.047462,\Rx:=0.000000,\Ry:=-8.273467),vel1,zoneval,Extruder\WObj:=Workobject_1;
MoveL RelTool (p1,20.500000,4.500000,9.656101,\Rx:=0.000000,\Ry:=-11.659006),vel1,zoneval,Extruder\WObj:=Workobject_1;
MoveL RelTool (p1,18.000000,4.500000,7.667393,\Rx:=0.000000,\Ry:=-2.952187),vel1,zoneval,Extruder\WObj:=Workobject_1;
MoveL RelTool (p1,15.500000,4.500000,7.500000,\Rx:=0.000000,\Ry:=0.000000),vel1,zoneval,Extruder\WObj:=Workobject_1;
MoveL RelTool (p1,13.000000,4.500000,7.500000,\Rx:=0.000000,\Ry:=0.000000),vel1,zoneval,Extruder\WObj:=Workobject_1;
MoveL RelTool (p1,10.500000,4.500000,7.500000,\Rx:=0.000000,\Ry:=0.000000),vel1,zoneval,Extruder\WObj:=Workobject_1;
MoveL RelTool (p1,8.000000,4.500000,7.500000,\Rx:=0.000000,\Ry:=0.000000),vel1,zoneval,Extruder\WObj:=Workobject_1;
MoveL RelTool (p1,5.500000,4.500000,7.500000,\Rx:=0.000000,\Ry:=0.000000),vel1,zoneval,Extruder\WObj:=Workobject_1;
MoveL RelTool (p1,3.000000,4.500000,7.500000,\Rx:=0.000000,\Ry:=0.000000),vel1,zoneval,Extruder\WObj:=Workobject_1;
MoveL RelTool (p1,5.000000,5.000000,7.500000,\Rx:=0.000000,\Ry:=-0.000000),vel1,zoneval,Extruder\WObj:=Workobject_1;
MoveL RelTool (p1,7.500000,5.000000,7.500000,\Rx:=0.000000,\Ry:=-0.000000),vel1,zoneval,Extruder\WObj:=Workobject_1;
MoveL RelTool (p1,10.000000,5.000000,7.500000,\Rx:=0.000000,\Ry:=-0.000000),vel1,zoneval,Extruder\WObj:=Workobject_1;
MoveL RelTool (p1,12.500000,5.000000,7.500000,\Rx:=0.000000,\Ry:=-0.000000),vel1,zoneval,Extruder\WObj:=Workobject_1;
MoveL RelTool (p1,15.000000,5.000000,7.500000,\Rx:=0.000000,\Ry:=-0.000000),vel1,zoneval,Extruder\WObj:=Workobject_1;
MoveL RelTool (p1,17.500000,5.000000,7.549338,\Rx:=0.000000,\Ry:=-2.952187),vel1,zoneval,Extruder\WObj:=Workobject_1;
MoveL RelTool (p1,20.000000,5.000000,9.005299,\Rx:=0.000000,\Ry:=-11.662773),vel1,zoneval,Extruder\WObj:=Workobject_1;
MoveL RelTool (p1,22.500000,5.000000,11.668030,\Rx:=0.000000,\Ry:=-8.284974),vel1,zoneval,Extruder\WObj:=Workobject_1;
MoveL RelTool (p1,25.000000,5.000000,13.346803,\Rx:=0.000000,\Ry:=-6.524894),vel1,zoneval,Extruder\WObj:=Workobject_1;
MoveL RelTool (p1,27.500000,5.000000,14.584021,\Rx:=0.000000,\Ry:=-5.324828),vel1,zoneval,Extruder\WObj:=Workobject_1;
MoveL RelTool (p1,30.000000,5.000000,15.528017,\Rx:=0.000000,\Ry:=-4.264941),vel1,zoneval,Extruder\WObj:=Workobject_1;
MoveL RelTool (p1,32.500000,5.000000,16.249855,\Rx:=0.000000,\Ry:=-3.285097),vel1,zoneval,Extruder\WObj:=Workobject_1;
MoveL RelTool (p1,35.000000,5.000000,16.779222,\Rx:=0.000000,\Ry:=-2.343931),vel1,zoneval,Extruder\WObj:=Workobject_1;
MoveL RelTool (p1,37.500000,5.000000,17.156067,\Rx:=0.000000,\Ry:=-1.457462),vel1,zoneval,Extruder\WObj:=Workobject_1;
MoveL RelTool (p1,40.000000,5.000000,17.391417,\Rx:=0.000000,\Ry:=-0.607859),vel1,zoneval,Extruder\WObj:=Workobject_1;
MoveL RelTool (p1,42.500000,5.000000,17.494222,\Rx:=0.000000,\Ry:=0.236465),vel1,zoneval,Extruder\WObj:=Workobject_1;
MoveL RelTool (p1,45.000000,5.000000,17.447787,\Rx:=0.000000,\Ry:=0.623075),vel1,zoneval,Extruder\WObj:=Workobject_1;
MoveL RelTool (p1,47.500000,5.000000,17.254470,\Rx:=0.000000,\Ry:=1.077014),vel1,zoneval,Extruder\WObj:=Workobject_1;
MoveL RelTool (p1,50.000000,5.000000,16.924208,\Rx:=0.000000,\Ry:=1.924676),vel1,zoneval,Extruder\WObj:=Workobject_1;
MoveL RelTool (p1,52.500000,5.000000,16.444808,\Rx:=0.000000,\Ry:=2.815279),vel1,zoneval,Extruder\WObj:=Workobject_1;
MoveL RelTool (p1,55.000000,5.000000,15.785061,\Rx:=0.000000,\Ry:=3.755557),vel1,zoneval,Extruder\WObj:=Workobject_1;
MoveL RelTool (p1,57.500000,5.000000,14.926118,\Rx:=0.000000,\Ry:=4.733408),vel1,zoneval,Extruder\WObj:=Workobject_1;
MoveL RelTool (p1,60.000000,5.000000,13.804534,\Rx:=0.000000,\Ry:=5.834401),vel1,zoneval,Extruder\WObj:=Workobject_1;
MoveL RelTool (p1,62.500000,5.000000,12.295179,\Rx:=0.000000,\Ry:=8.283792),vel1,zoneval,Extruder\WObj:=Workobject_1;
MoveL RelTool (p1,65.000000,5.000000,10.046181,\Rx:=0.000000,\Ry:=11.396766),vel1,zoneval,Extruder\WObj:=Workobject_1;
MoveL RelTool (p1,67.500000,5.000000,7.780757,\Rx:=0.000000,\Ry:=3.821551),vel1,zoneval,Extruder\WObj:=Workobject_1;
MoveL RelTool (p1,70.000000,5.000000,7.500000,\Rx:=0.000000,\Ry:=-0.000000),vel1,zoneval,Extruder\WObj:=Workobject_1;
MoveL RelTool (p1,72.500000,5.000000,7.500000,\Rx:=0.000000,\Ry:=-0.000000),vel1,zoneval,Extruder\WObj:=Workobject_1;
MoveL RelTool (p1,75.000000,5.000000,7.500000,\Rx:=0.000000,\Ry:=-0.000000),vel1,zoneval,Extruder\WObj:=Workobject_1;
MoveL RelTool (p1,77.500000,5.000000,7.500000,\Rx:=0.000000,\Ry:=-0.000000),vel1,zoneval,Extruder\WObj:=Workobject_1;
MoveL RelTool (p1,80.000000,5.000000,7.500000,\Rx:=0.000000,\Ry:=-0.000000),vel1,zoneval,Extruder\WObj:=Workobject_1;
MoveL RelTool (p1,82.500000,5.000000,7.500000,\Rx:=0.000000,\Ry:=-0.000000),vel1,zoneval,Extruder\WObj:=Workobject_1;
MoveL RelTool (p1,80.500000,5.500000,7.500000,\Rx:=0.000000,\Ry:=0.000000),vel1,zoneval,Extruder\WObj:=Workobject_1;
MoveL RelTool (p1,78.000000,5.500000,7.500000,\Rx:=0.000000,\Ry:=0.000000),vel1,zoneval,Extruder\WObj:=Workobject_1;
MoveL RelTool (p1,75.500000,5.500000,7.500000,\Rx:=0.000000,\Ry:=0.000000),vel1,zoneval,Extruder\WObj:=Workobject_1;
MoveL RelTool (p1,73.000000,5.500000,7.500000,\Rx:=0.000000,\Ry:=0.000000),vel1,zoneval,Extruder\WObj:=Workobject_1;
MoveL RelTool (p1,70.500000,5.500000,7.500000,\Rx:=0.000000,\Ry:=0.000000),vel1,zoneval,Extruder\WObj:=Workobject_1;
MoveL RelTool (p1,68.000000,5.500000,7.626010,\Rx:=0.000000,\Ry:=3.821551),vel1,zoneval,Extruder\WObj:=Workobject_1;
MoveL RelTool (p1,65.500000,5.500000,9.423912,\Rx:=0.000000,\Ry:=11.396766),vel1,zoneval,Extruder\WObj:=Workobject_1;
MoveL RelTool (p1,63.000000,5.500000,11.915624,\Rx:=0.000000,\Ry:=8.283792),vel1,zoneval,Extruder\WObj:=Workobject_1;
MoveL RelTool (p1,60.500000,5.500000,13.557752,\Rx:=0.000000,\Ry:=5.843574),vel1,zoneval,Extruder\WObj:=Workobject_1;
MoveL RelTool (p1,58.000000,5.500000,14.731880,\Rx:=0.000000,\Ry:=4.733408),vel1,zoneval,Extruder\WObj:=Workobject_1;
MoveL RelTool (p1,55.500000,5.500000,15.633168,\Rx:=0.000000,\Ry:=3.755557),vel1,zoneval,Extruder\WObj:=Workobject_1;
MoveL RelTool (p1,53.000000,5.500000,16.333395,\Rx:=0.000000,\Ry:=2.815279),vel1,zoneval,Extruder\WObj:=Workobject_1;
MoveL RelTool (p1,50.500000,5.500000,16.848523,\Rx:=0.000000,\Ry:=1.924676),vel1,zoneval,Extruder\WObj:=Workobject_1;
MoveL RelTool (p1,48.000000,5.500000,17.212898,\Rx:=0.000000,\Ry:=1.077014),vel1,zoneval,Extruder\WObj:=Workobject_1;
MoveL RelTool (p1,45.500000,5.500000,17.423561,\Rx:=0.000000,\Ry:=0.641125),vel1,zoneval,Extruder\WObj:=Workobject_1;
MoveL RelTool (p1,43.000000,5.500000,17.485908,\Rx:=0.000000,\Ry:=0.213870),vel1,zoneval,Extruder\WObj:=Workobject_1;
MoveL RelTool (p1,40.500000,5.500000,17.416204,\Rx:=0.000000,\Ry:=-0.607859),vel1,zoneval,Extruder\WObj:=Workobject_1;
MoveL RelTool (p1,38.000000,5.500000,17.214218,\Rx:=0.000000,\Ry:=-1.457462),vel1,zoneval,Extruder\WObj:=Workobject_1;
MoveL RelTool (p1,35.500000,5.500000,16.872573,\Rx:=0.000000,\Ry:=-2.343931),vel1,zoneval,Extruder\WObj:=Workobject_1;
MoveL RelTool (p1,33.000000,5.500000,16.382860,\Rx:=0.000000,\Ry:=-3.285097),vel1,zoneval,Extruder\WObj:=Workobject_1;
MoveL RelTool (p1,30.500000,5.500000,15.702416,\Rx:=0.000000,\Ry:=-4.264941),vel1,zoneval,Extruder\WObj:=Workobject_1;
MoveL RelTool (p1,28.000000,5.500000,14.807149,\Rx:=0.000000,\Ry:=-5.329822),vel1,zoneval,Extruder\WObj:=Workobject_1;
MoveL RelTool (p1,25.500000,5.500000,13.629250,\Rx:=0.000000,\Ry:=-6.524894),vel1,zoneval,Extruder\WObj:=Workobject_1;
MoveL RelTool (p1,23.000000,5.500000,12.049908,\Rx:=0.000000,\Ry:=-8.296465),vel1,zoneval,Extruder\WObj:=Workobject_1;
MoveL RelTool (p1,20.500000,5.500000,9.656898,\Rx:=0.000000,\Ry:=-11.666537),vel1,zoneval,Extruder\WObj:=Workobject_1;
MoveL RelTool (p1,18.000000,5.500000,7.667393,\Rx:=0.000000,\Ry:=-2.952187),vel1,zoneval,Extruder\WObj:=Workobject_1;
MoveL RelTool (p1,15.500000,5.500000,7.500000,\Rx:=0.000000,\Ry:=0.000000),vel1,zoneval,Extruder\WObj:=Workobject_1;
MoveL RelTool (p1,13.000000,5.500000,7.500000,\Rx:=0.000000,\Ry:=0.000000),vel1,zoneval,Extruder\WObj:=Workobject_1;
MoveL RelTool (p1,10.500000,5.500000,7.500000,\Rx:=0.000000,\Ry:=0.000000),vel1,zoneval,Extruder\WObj:=Workobject_1;
MoveL RelTool (p1,8.000000,5.500000,7.500000,\Rx:=0.000000,\Ry:=0.000000),vel1,zoneval,Extruder\WObj:=Workobject_1;
MoveL RelTool (p1,5.500000,5.500000,7.500000,\Rx:=0.000000,\Ry:=0.000000),vel1,zoneval,Extruder\WObj:=Workobject_1;
MoveL RelTool (p1,3.000000,5.500000,7.500000,\Rx:=0.000000,\Ry:=0.000000),vel1,zoneval,Extruder\WObj:=Workobject_1;
MoveL RelTool (p1,5.000000,6.000000,7.500000,\Rx:=0.000000,\Ry:=-0.000000),vel1,zoneval,Extruder\WObj:=Workobject_1;
MoveL RelTool (p1,7.500000,6.000000,7.500000,\Rx:=0.000000,\Ry:=-0.000000),vel1,zoneval,Extruder\WObj:=Workobject_1;
MoveL RelTool (p1,10.000000,6.000000,7.500000,\Rx:=0.000000,\Ry:=-0.000000),vel1,zoneval,Extruder\WObj:=Workobject_1;
MoveL RelTool (p1,12.500000,6.000000,7.500000,\Rx:=0.000000,\Ry:=-0.000000),vel1,zoneval,Extruder\WObj:=Workobject_1;
MoveL RelTool (p1,15.000000,6.000000,7.500000,\Rx:=0.000000,\Ry:=-0.000000),vel1,zoneval,Extruder\WObj:=Workobject_1;
MoveL RelTool (p1,17.500000,6.000000,7.549338,\Rx:=0.000000,\Ry:=-2.952187),vel1,zoneval,Extruder\WObj:=Workobject_1;
MoveL RelTool (p1,20.000000,6.000000,9.005299,\Rx:=0.000000,\Ry:=-11.670299),vel1,zoneval,Extruder\WObj:=Workobject_1;
MoveL RelTool (p1,22.500000,6.000000,11.669050,\Rx:=0.000000,\Ry:=-8.307940),vel1,zoneval,Extruder\WObj:=Workobject_1;
MoveL RelTool (p1,25.000000,6.000000,13.349098,\Rx:=0.000000,\Ry:=-6.524894),vel1,zoneval,Extruder\WObj:=Workobject_1;
MoveL RelTool (p1,27.500000,6.000000,14.585378,\Rx:=0.000000,\Ry:=-5.334815),vel1,zoneval,Extruder\WObj:=Workobject_1;
MoveL RelTool (p1,30.000000,6.000000,15.528730,\Rx:=0.000000,\Ry:=-4.264941),vel1,zoneval,Extruder\WObj:=Workobject_1;
MoveL RelTool (p1,32.500000,6.000000,16.251973,\Rx:=0.000000,\Ry:=-3.285097),vel1,zoneval,Extruder\WObj:=Workobject_1;
MoveL RelTool (p1,35.000000,6.000000,16.779725,\Rx:=0.000000,\Ry:=-2.343931),vel1,zoneval,Extruder\WObj:=Workobject_1;
MoveL RelTool (p1,37.500000,6.000000,17.157397,\Rx:=0.000000,\Ry:=-1.457462),vel1,zoneval,Extruder\WObj:=Workobject_1;
MoveL RelTool (p1,40.000000,6.000000,17.393213,\Rx:=0.000000,\Ry:=-0.607859),vel1,zoneval,Extruder\WObj:=Workobject_1;
MoveL RelTool (p1,42.500000,6.000000,17.494193,\Rx:=0.000000,\Ry:=0.186191),vel1,zoneval,Extruder\WObj:=Workobject_1;
MoveL RelTool (p1,45.000000,6.000000,17.448786,\Rx:=0.000000,\Ry:=0.635132),vel1,zoneval,Extruder\WObj:=Workobject_1;
MoveL RelTool (p1,47.500000,6.000000,17.256117,\Rx:=0.000000,\Ry:=1.077014),vel1,zoneval,Extruder\WObj:=Workobject_1;
MoveL RelTool (p1,50.000000,6.000000,16.925163,\Rx:=0.000000,\Ry:=1.924676),vel1,zoneval,Extruder\WObj:=Workobject_1;
MoveL RelTool (p1,52.500000,6.000000,16.446769,\Rx:=0.000000,\Ry:=2.815279),vel1,zoneval,Extruder\WObj:=Workobject_1;
MoveL RelTool (p1,55.000000,6.000000,15.785097,\Rx:=0.000000,\Ry:=3.755557),vel1,zoneval,Extruder\WObj:=Workobject_1;
MoveL RelTool (p1,57.500000,6.000000,14.927532,\Rx:=0.000000,\Ry:=4.733408),vel1,zoneval,Extruder\WObj:=Workobject_1;
MoveL RelTool (p1,60.000000,6.000000,13.805116,\Rx:=0.000000,\Ry:=5.852740),vel1,zoneval,Extruder\WObj:=Workobject_1;
MoveL RelTool (p1,62.500000,6.000000,12.297232,\Rx:=0.000000,\Ry:=8.283792),vel1,zoneval,Extruder\WObj:=Workobject_1;
MoveL RelTool (p1,65.000000,6.000000,10.049197,\Rx:=0.000000,\Ry:=11.396766),vel1,zoneval,Extruder\WObj:=Workobject_1;
MoveL RelTool (p1,67.500000,6.000000,7.780757,\Rx:=0.000000,\Ry:=3.821551),vel1,zoneval,Extruder\WObj:=Workobject_1;
MoveL RelTool (p1,70.000000,6.000000,7.500000,\Rx:=0.000000,\Ry:=-0.000000),vel1,zoneval,Extruder\WObj:=Workobject_1;
MoveL RelTool (p1,72.500000,6.000000,7.500000,\Rx:=0.000000,\Ry:=-0.000000),vel1,zoneval,Extruder\WObj:=Workobject_1;
MoveL RelTool (p1,75.000000,6.000000,7.500000,\Rx:=0.000000,\Ry:=-0.000000),vel1,zoneval,Extruder\WObj:=Workobject_1;
MoveL RelTool (p1,77.500000,6.000000,7.500000,\Rx:=0.000000,\Ry:=-0.000000),vel1,zoneval,Extruder\WObj:=Workobject_1;
MoveL RelTool (p1,80.000000,6.000000,7.500000,\Rx:=0.000000,\Ry:=-0.000000),vel1,zoneval,Extruder\WObj:=Workobject_1;
MoveL RelTool (p1,82.500000,6.000000,7.500000,\Rx:=0.000000,\Ry:=-0.000000),vel1,zoneval,Extruder\WObj:=Workobject_1;
MoveL RelTool (p1,80.500000,6.500000,7.500000,\Rx:=0.000000,\Ry:=0.000000),vel1,zoneval,Extruder\WObj:=Workobject_1;
MoveL RelTool (p1,78.000000,6.500000,7.500000,\Rx:=0.000000,\Ry:=0.000000),vel1,zoneval,Extruder\WObj:=Workobject_1;
MoveL RelTool (p1,75.500000,6.500000,7.500000,\Rx:=0.000000,\Ry:=0.000000),vel1,zoneval,Extruder\WObj:=Workobject_1;
MoveL RelTool (p1,73.000000,6.500000,7.500000,\Rx:=0.000000,\Ry:=0.000000),vel1,zoneval,Extruder\WObj:=Workobject_1;
MoveL RelTool (p1,70.500000,6.500000,7.500000,\Rx:=0.000000,\Ry:=0.000000),vel1,zoneval,Extruder\WObj:=Workobject_1;
MoveL RelTool (p1,68.000000,6.500000,7.626010,\Rx:=0.000000,\Ry:=3.821551),vel1,zoneval,Extruder\WObj:=Workobject_1;
MoveL RelTool (p1,65.500000,6.500000,9.426927,\Rx:=0.000000,\Ry:=11.396766),vel1,zoneval,Extruder\WObj:=Workobject_1;
MoveL RelTool (p1,63.000000,6.500000,11.917678,\Rx:=0.000000,\Ry:=8.283792),vel1,zoneval,Extruder\WObj:=Workobject_1;
MoveL RelTool (p1,60.500000,6.500000,13.557439,\Rx:=0.000000,\Ry:=5.861900),vel1,zoneval,Extruder\WObj:=Workobject_1;
MoveL RelTool (p1,58.000000,6.500000,14.733293,\Rx:=0.000000,\Ry:=4.733408),vel1,zoneval,Extruder\WObj:=Workobject_1;
MoveL RelTool (p1,55.500000,6.500000,15.633204,\Rx:=0.000000,\Ry:=3.755557),vel1,zoneval,Extruder\WObj:=Workobject_1;
MoveL RelTool (p1,53.000000,6.500000,16.335356,\Rx:=0.000000,\Ry:=2.815279),vel1,zoneval,Extruder\WObj:=Workobject_1;
MoveL RelTool (p1,50.500000,6.500000,16.849478,\Rx:=0.000000,\Ry:=1.924676),vel1,zoneval,Extruder\WObj:=Workobject_1;
MoveL RelTool (p1,48.000000,6.500000,17.214545,\Rx:=0.000000,\Ry:=1.077014),vel1,zoneval,Extruder\WObj:=Workobject_1;
MoveL RelTool (p1,45.500000,6.500000,17.424086,\Rx:=0.000000,\Ry:=0.623872),vel1,zoneval,Extruder\WObj:=Workobject_1;
MoveL RelTool (p1,43.000000,6.500000,17.487853,\Rx:=0.000000,\Ry:=0.158511),vel1,zoneval,Extruder\WObj:=Workobject_1;
MoveL RelTool (p1,40.500000,6.500000,17.417999,\Rx:=0.000000,\Ry:=-0.607859),vel1,zoneval,Extruder\WObj:=Workobject_1;
MoveL RelTool (p1,38.000000,6.500000,17.215548,\Rx:=0.000000,\Ry:=-1.457462),vel1,zoneval,Extruder\WObj:=Workobject_1;
MoveL RelTool (p1,35.500000,6.500000,16.873076,\Rx:=0.000000,\Ry:=-2.343931),vel1,zoneval,Extruder\WObj:=Workobject_1;
MoveL RelTool (p1,33.000000,6.500000,16.384754,\Rx:=0.000000,\Ry:=-3.279770),vel1,zoneval,Extruder\WObj:=Workobject_1;
MoveL RelTool (p1,30.500000,6.500000,15.703129,\Rx:=0.000000,\Ry:=-4.264941),vel1,zoneval,Extruder\WObj:=Workobject_1;
MoveL RelTool (p1,28.000000,6.500000,14.808976,\Rx:=0.000000,\Ry:=-5.339805),vel1,zoneval,Extruder\WObj:=Workobject_1;
MoveL RelTool (p1,25.500000,6.500000,13.631544,\Rx:=0.000000,\Ry:=-6.524894),vel1,zoneval,Extruder\WObj:=Workobject_1;
MoveL RelTool (p1,23.000000,6.500000,12.052355,\Rx:=0.000000,\Ry:=-8.319400),vel1,zoneval,Extruder\WObj:=Workobject_1;
MoveL RelTool (p1,20.500000,6.500000,9.657696,\Rx:=0.000000,\Ry:=-11.674057),vel1,zoneval,Extruder\WObj:=Workobject_1;
MoveL RelTool (p1,18.000000,6.500000,7.667393,\Rx:=0.000000,\Ry:=-2.952187),vel1,zoneval,Extruder\WObj:=Workobject_1;
MoveL RelTool (p1,15.500000,6.500000,7.500000,\Rx:=0.000000,\Ry:=0.000000),vel1,zoneval,Extruder\WObj:=Workobject_1;
MoveL RelTool (p1,13.000000,6.500000,7.500000,\Rx:=0.000000,\Ry:=0.000000),vel1,zoneval,Extruder\WObj:=Workobject_1;
MoveL RelTool (p1,10.500000,6.500000,7.500000,\Rx:=0.000000,\Ry:=0.000000),vel1,zoneval,Extruder\WObj:=Workobject_1;
MoveL RelTool (p1,8.000000,6.500000,7.500000,\Rx:=0.000000,\Ry:=0.000000),vel1,zoneval,Extruder\WObj:=Workobject_1;
MoveL RelTool (p1,5.500000,6.500000,7.500000,\Rx:=0.000000,\Ry:=0.000000),vel1,zoneval,Extruder\WObj:=Workobject_1;
MoveL RelTool (p1,3.000000,6.500000,7.500000,\Rx:=0.000000,\Ry:=0.000000),vel1,zoneval,Extruder\WObj:=Workobject_1;
MoveL RelTool (p1,5.000000,7.000000,7.500000,\Rx:=0.000000,\Ry:=-0.000000),vel1,zoneval,Extruder\WObj:=Workobject_1;
MoveL RelTool (p1,7.500000,7.000000,7.500000,\Rx:=0.000000,\Ry:=-0.000000),vel1,zoneval,Extruder\WObj:=Workobject_1;
MoveL RelTool (p1,10.000000,7.000000,7.500000,\Rx:=0.000000,\Ry:=-0.000000),vel1,zoneval,Extruder\WObj:=Workobject_1;
MoveL RelTool (p1,12.500000,7.000000,7.500000,\Rx:=0.000000,\Ry:=-0.000000),vel1,zoneval,Extruder\WObj:=Workobject_1;
MoveL RelTool (p1,15.000000,7.000000,7.500000,\Rx:=0.000000,\Ry:=-0.000000),vel1,zoneval,Extruder\WObj:=Workobject_1;
MoveL RelTool (p1,17.500000,7.000000,7.549338,\Rx:=0.000000,\Ry:=-2.952187),vel1,zoneval,Extruder\WObj:=Workobject_1;
MoveL RelTool (p1,20.000000,7.000000,9.005299,\Rx:=0.000000,\Ry:=-11.677813),vel1,zoneval,Extruder\WObj:=Workobject_1;
MoveL RelTool (p1,22.500000,7.000000,11.670070,\Rx:=0.000000,\Ry:=-8.330843),vel1,zoneval,Extruder\WObj:=Workobject_1;
MoveL RelTool (p1,25.000000,7.000000,13.351393,\Rx:=0.000000,\Ry:=-6.524894),vel1,zoneval,Extruder\WObj:=Workobject_1;
MoveL RelTool (p1,27.500000,7.000000,14.586735,\Rx:=0.000000,\Ry:=-5.344794),vel1,zoneval,Extruder\WObj:=Workobject_1;
MoveL RelTool (p1,30.000000,7.000000,15.529443,\Rx:=0.000000,\Ry:=-4.264941),vel1,zoneval,Extruder\WObj:=Workobject_1;
MoveL RelTool (p1,32.500000,7.000000,16.254090,\Rx:=0.000000,\Ry:=-3.251791),vel1,zoneval,Extruder\WObj:=Workobject_1;
MoveL RelTool (p1,35.000000,7.000000,16.780227,\Rx:=0.000000,\Ry:=-2.371315),vel1,zoneval,Extruder\WObj:=Workobject_1;
MoveL RelTool (p1,37.500000,7.000000,17.158727,\Rx:=0.000000,\Ry:=-1.457462),vel1,zoneval,Extruder\WObj:=Workobject_1;
MoveL RelTool (p1,40.000000,7.000000,17.395009,\Rx:=0.000000,\Ry:=-0.607859),vel1,zoneval,Extruder\WObj:=Workobject_1;
MoveL RelTool (p1,42.500000,7.000000,17.493963,\Rx:=0.000000,\Ry:=0.130829),vel1,zoneval,Extruder\WObj:=Workobject_1;
MoveL RelTool (p1,45.000000,7.000000,17.448423,\Rx:=0.000000,\Ry:=0.612611),vel1,zoneval,Extruder\WObj:=Workobject_1;
MoveL RelTool (p1,47.500000,7.000000,17.257764,\Rx:=0.000000,\Ry:=1.091787),vel1,zoneval,Extruder\WObj:=Workobject_1;
MoveL RelTool (p1,50.000000,7.000000,16.926119,\Rx:=0.000000,\Ry:=1.924676),vel1,zoneval,Extruder\WObj:=Workobject_1;
MoveL RelTool (p1,52.500000,7.000000,16.448730,\Rx:=0.000000,\Ry:=2.815279),vel1,zoneval,Extruder\WObj:=Workobject_1;
MoveL RelTool (p1,55.000000,7.000000,15.785134,\Rx:=0.000000,\Ry:=3.755557),vel1,zoneval,Extruder\WObj:=Workobject_1;
MoveL RelTool (p1,57.500000,7.000000,14.928946,\Rx:=0.000000,\Ry:=4.733408),vel1,zoneval,Extruder\WObj:=Workobject_1;
MoveL RelTool (p1,60.000000,7.000000,13.805699,\Rx:=0.000000,\Ry:=5.871053),vel1,zoneval,Extruder\WObj:=Workobject_1;
MoveL RelTool (p1,62.500000,7.000000,12.299286,\Rx:=0.000000,\Ry:=8.283792),vel1,zoneval,Extruder\WObj:=Workobject_1;
MoveL RelTool (p1,65.000000,7.000000,10.052213,\Rx:=0.000000,\Ry:=11.397950),vel1,zoneval,Extruder\WObj:=Workobject_1;
MoveL RelTool (p1,67.500000,7.000000,7.780757,\Rx:=0.000000,\Ry:=3.821551),vel1,zoneval,Extruder\WObj:=Workobject_1;
MoveL RelTool (p1,70.000000,7.000000,7.500000,\Rx:=0.000000,\Ry:=-0.000000),vel1,zoneval,Extruder\WObj:=Workobject_1;
MoveL RelTool (p1,72.500000,7.000000,7.500000,\Rx:=0.000000,\Ry:=-0.000000),vel1,zoneval,Extruder\WObj:=Workobject_1;
MoveL RelTool (p1,75.000000,7.000000,7.500000,\Rx:=0.000000,\Ry:=-0.000000),vel1,zoneval,Extruder\WObj:=Workobject_1;
MoveL RelTool (p1,77.500000,7.000000,7.500000,\Rx:=0.000000,\Ry:=-0.000000),vel1,zoneval,Extruder\WObj:=Workobject_1;
MoveL RelTool (p1,80.000000,7.000000,7.500000,\Rx:=0.000000,\Ry:=-0.000000),vel1,zoneval,Extruder\WObj:=Workobject_1;
MoveL RelTool (p1,82.500000,7.000000,7.500000,\Rx:=0.000000,\Ry:=-0.000000),vel1,zoneval,Extruder\WObj:=Workobject_1;
MoveL RelTool (p1,80.500000,7.500000,7.500000,\Rx:=0.000000,\Ry:=0.000000),vel1,zoneval,Extruder\WObj:=Workobject_1;
MoveL RelTool (p1,78.000000,7.500000,7.500000,\Rx:=0.000000,\Ry:=0.000000),vel1,zoneval,Extruder\WObj:=Workobject_1;
MoveL RelTool (p1,75.500000,7.500000,7.500000,\Rx:=0.000000,\Ry:=0.000000),vel1,zoneval,Extruder\WObj:=Workobject_1;
MoveL RelTool (p1,73.000000,7.500000,7.500000,\Rx:=0.000000,\Ry:=0.000000),vel1,zoneval,Extruder\WObj:=Workobject_1;
MoveL RelTool (p1,70.500000,7.500000,7.500000,\Rx:=0.000000,\Ry:=0.000000),vel1,zoneval,Extruder\WObj:=Workobject_1;
MoveL RelTool (p1,68.000000,7.500000,7.626010,\Rx:=0.000000,\Ry:=3.821551),vel1,zoneval,Extruder\WObj:=Workobject_1;
MoveL RelTool (p1,65.500000,7.500000,9.428317,\Rx:=0.000000,\Ry:=11.412945),vel1,zoneval,Extruder\WObj:=Workobject_1;
MoveL RelTool (p1,63.000000,7.500000,11.919731,\Rx:=0.000000,\Ry:=8.274330),vel1,zoneval,Extruder\WObj:=Workobject_1;
MoveL RelTool (p1,60.500000,7.500000,13.557125,\Rx:=0.000000,\Ry:=5.880200),vel1,zoneval,Extruder\WObj:=Workobject_1;
MoveL RelTool (p1,58.000000,7.500000,14.734707,\Rx:=0.000000,\Ry:=4.733408),vel1,zoneval,Extruder\WObj:=Workobject_1;
MoveL RelTool (p1,55.500000,7.500000,15.634255,\Rx:=0.000000,\Ry:=3.731872),vel1,zoneval,Extruder\WObj:=Workobject_1;
MoveL RelTool (p1,53.000000,7.500000,16.337317,\Rx:=0.000000,\Ry:=2.815279),vel1,zoneval,Extruder\WObj:=Workobject_1;
MoveL RelTool (p1,50.500000,7.500000,16.850433,\Rx:=0.000000,\Ry:=1.924676),vel1,zoneval,Extruder\WObj:=Workobject_1;
MoveL RelTool (p1,48.000000,7.500000,17.214466,\Rx:=0.000000,\Ry:=1.120627),vel1,zoneval,Extruder\WObj:=Workobject_1;
MoveL RelTool (p1,45.500000,7.500000,17.424610,\Rx:=0.000000,\Ry:=0.601349),vel1,zoneval,Extruder\WObj:=Workobject_1;
MoveL RelTool (p1,43.000000,7.500000,17.489798,\Rx:=0.000000,\Ry:=0.103145),vel1,zoneval,Extruder\WObj:=Workobject_1;
MoveL RelTool (p1,40.500000,7.500000,17.419795,\Rx:=0.000000,\Ry:=-0.607859),vel1,zoneval,Extruder\WObj:=Workobject_1;
MoveL RelTool (p1,38.000000,7.500000,17.216878,\Rx:=0.000000,\Ry:=-1.457462),vel1,zoneval,Extruder\WObj:=Workobject_1;
MoveL RelTool (p1,35.500000,7.500000,16.875872,\Rx:=0.000000,\Ry:=-2.400326),vel1,zoneval,Extruder\WObj:=Workobject_1;
MoveL RelTool (p1,33.000000,7.500000,16.384523,\Rx:=0.000000,\Ry:=-3.223780),vel1,zoneval,Extruder\WObj:=Workobject_1;
MoveL RelTool (p1,30.500000,7.500000,15.703842,\Rx:=0.000000,\Ry:=-4.264941),vel1,zoneval,Extruder\WObj:=Workobject_1;
MoveL RelTool (p1,28.000000,7.500000,14.810802,\Rx:=0.000000,\Ry:=-5.349782),vel1,zoneval,Extruder\WObj:=Workobject_1;
MoveL RelTool (p1,25.500000,7.500000,13.633839,\Rx:=0.000000,\Ry:=-6.524894),vel1,zoneval,Extruder\WObj:=Workobject_1;
MoveL RelTool (p1,23.000000,7.500000,12.054801,\Rx:=0.000000,\Ry:=-8.342271),vel1,zoneval,Extruder\WObj:=Workobject_1;
MoveL RelTool (p1,20.500000,7.500000,9.658493,\Rx:=0.000000,\Ry:=-11.681565),vel1,zoneval,Extruder\WObj:=Workobject_1;
MoveL RelTool (p1,18.000000,7.500000,7.667393,\Rx:=0.000000,\Ry:=-2.952187),vel1,zoneval,Extruder\WObj:=Workobject_1;
MoveL RelTool (p1,15.500000,7.500000,7.500000,\Rx:=0.000000,\Ry:=0.000000),vel1,zoneval,Extruder\WObj:=Workobject_1;
MoveL RelTool (p1,13.000000,7.500000,7.500000,\Rx:=0.000000,\Ry:=0.000000),vel1,zoneval,Extruder\WObj:=Workobject_1;
MoveL RelTool (p1,10.500000,7.500000,7.500000,\Rx:=0.000000,\Ry:=0.000000),vel1,zoneval,Extruder\WObj:=Workobject_1;
MoveL RelTool (p1,8.000000,7.500000,7.500000,\Rx:=0.000000,\Ry:=0.000000),vel1,zoneval,Extruder\WObj:=Workobject_1;
MoveL RelTool (p1,5.500000,7.500000,7.500000,\Rx:=0.000000,\Ry:=0.000000),vel1,zoneval,Extruder\WObj:=Workobject_1;
MoveL RelTool (p1,3.000000,7.500000,7.500000,\Rx:=0.000000,\Ry:=0.000000),vel1,zoneval,Extruder\WObj:=Workobject_1;
MoveL RelTool (p1,5.000000,8.000000,7.500000,\Rx:=0.000000,\Ry:=-0.000000),vel1,zoneval,Extruder\WObj:=Workobject_1;
MoveL RelTool (p1,7.500000,8.000000,7.500000,\Rx:=0.000000,\Ry:=-0.000000),vel1,zoneval,Extruder\WObj:=Workobject_1;
MoveL RelTool (p1,10.000000,8.000000,7.500000,\Rx:=0.000000,\Ry:=-0.000000),vel1,zoneval,Extruder\WObj:=Workobject_1;
MoveL RelTool (p1,12.500000,8.000000,7.500000,\Rx:=0.000000,\Ry:=-0.000000),vel1,zoneval,Extruder\WObj:=Workobject_1;
MoveL RelTool (p1,15.000000,8.000000,7.500000,\Rx:=0.000000,\Ry:=-0.000000),vel1,zoneval,Extruder\WObj:=Workobject_1;
MoveL RelTool (p1,17.500000,8.000000,7.549338,\Rx:=0.000000,\Ry:=-2.952187),vel1,zoneval,Extruder\WObj:=Workobject_1;
MoveL RelTool (p1,20.000000,8.000000,9.005299,\Rx:=0.000000,\Ry:=-11.685315),vel1,zoneval,Extruder\WObj:=Workobject_1;
MoveL RelTool (p1,22.500000,8.000000,11.671090,\Rx:=0.000000,\Ry:=-8.353683),vel1,zoneval,Extruder\WObj:=Workobject_1;
MoveL RelTool (p1,25.000000,8.000000,13.353687,\Rx:=0.000000,\Ry:=-6.524894),vel1,zoneval,Extruder\WObj:=Workobject_1;
MoveL RelTool (p1,27.500000,8.000000,14.588092,\Rx:=0.000000,\Ry:=-5.354767),vel1,zoneval,Extruder\WObj:=Workobject_1;
MoveL RelTool (p1,30.000000,8.000000,15.530156,\Rx:=0.000000,\Ry:=-4.264941),vel1,zoneval,Extruder\WObj:=Workobject_1;
MoveL RelTool (p1,32.500000,8.000000,16.256208,\Rx:=0.000000,\Ry:=-3.195738),vel1,zoneval,Extruder\WObj:=Workobject_1;
MoveL RelTool (p1,35.000000,8.000000,16.780730,\Rx:=0.000000,\Ry:=-2.429313),vel1,zoneval,Extruder\WObj:=Workobject_1;
MoveL RelTool (p1,37.500000,8.000000,17.160058,\Rx:=0.000000,\Ry:=-1.457462),vel1,zoneval,Extruder\WObj:=Workobject_1;
MoveL RelTool (p1,40.000000,8.000000,17.396804,\Rx:=0.000000,\Ry:=-0.607859),vel1,zoneval,Extruder\WObj:=Workobject_1;
MoveL RelTool (p1,42.500000,8.000000,17.493734,\Rx:=0.000000,\Ry:=0.075461),vel1,zoneval,Extruder\WObj:=Workobject_1;
MoveL RelTool (p1,45.000000,8.000000,17.448061,\Rx:=0.000000,\Ry:=0.590086),vel1,zoneval,Extruder\WObj:=Workobject_1;
MoveL RelTool (p1,47.500000,8.000000,17.259411,\Rx:=0.000000,\Ry:=1.149455),vel1,zoneval,Extruder\WObj:=Workobject_1;
MoveL RelTool (p1,50.000000,8.000000,16.927074,\Rx:=0.000000,\Ry:=1.924676),vel1,zoneval,Extruder\WObj:=Workobject_1;
MoveL RelTool (p1,52.500000,8.000000,16.450691,\Rx:=0.000000,\Ry:=2.815279),vel1,zoneval,Extruder\WObj:=Workobject_1;
MoveL RelTool (p1,55.000000,8.000000,15.785170,\Rx:=0.000000,\Ry:=3.693791),vel1,zoneval,Extruder\WObj:=Workobject_1;
MoveL RelTool (p1,57.500000,8.000000,14.930359,\Rx:=0.000000,\Ry:=4.733408),vel1,zoneval,Extruder\WObj:=Workobject_1;
MoveL RelTool (p1,60.000000,8.000000,13.806282,\Rx:=0.000000,\Ry:=5.889340),vel1,zoneval,Extruder\WObj:=Workobject_1;
MoveL RelTool (p1,62.500000,8.000000,12.300044,\Rx:=0.000000,\Ry:=8.262874),vel1,zoneval,Extruder\WObj:=Workobject_1;
MoveL RelTool (p1,65.000000,8.000000,10.055229,\Rx:=0.000000,\Ry:=11.427897),vel1,zoneval,Extruder\WObj:=Workobject_1;
MoveL RelTool (p1,67.500000,8.000000,7.780757,\Rx:=0.000000,\Ry:=3.821551),vel1,zoneval,Extruder\WObj:=Workobject_1;
MoveL RelTool (p1,70.000000,8.000000,7.500000,\Rx:=0.000000,\Ry:=-0.000000),vel1,zoneval,Extruder\WObj:=Workobject_1;
MoveL RelTool (p1,72.500000,8.000000,7.500000,\Rx:=0.000000,\Ry:=-0.000000),vel1,zoneval,Extruder\WObj:=Workobject_1;
MoveL RelTool (p1,75.000000,8.000000,7.500000,\Rx:=0.000000,\Ry:=-0.000000),vel1,zoneval,Extruder\WObj:=Workobject_1;
MoveL RelTool (p1,77.500000,8.000000,7.500000,\Rx:=0.000000,\Ry:=-0.000000),vel1,zoneval,Extruder\WObj:=Workobject_1;
MoveL RelTool (p1,80.000000,8.000000,7.500000,\Rx:=0.000000,\Ry:=-0.000000),vel1,zoneval,Extruder\WObj:=Workobject_1;
MoveL RelTool (p1,82.500000,8.000000,7.500000,\Rx:=0.000000,\Ry:=-0.000000),vel1,zoneval,Extruder\WObj:=Workobject_1;
MoveL RelTool (p1,80.500000,8.500000,7.500000,\Rx:=0.000000,\Ry:=0.000000),vel1,zoneval,Extruder\WObj:=Workobject_1;
MoveL RelTool (p1,78.000000,8.500000,7.500000,\Rx:=0.000000,\Ry:=0.000000),vel1,zoneval,Extruder\WObj:=Workobject_1;
MoveL RelTool (p1,75.500000,8.500000,7.500000,\Rx:=0.000000,\Ry:=0.000000),vel1,zoneval,Extruder\WObj:=Workobject_1;
MoveL RelTool (p1,73.000000,8.500000,7.500000,\Rx:=0.000000,\Ry:=0.000000),vel1,zoneval,Extruder\WObj:=Workobject_1;
MoveL RelTool (p1,70.500000,8.500000,7.500000,\Rx:=0.000000,\Ry:=0.000000),vel1,zoneval,Extruder\WObj:=Workobject_1;
MoveL RelTool (p1,68.000000,8.500000,7.626010,\Rx:=0.000000,\Ry:=3.821551),vel1,zoneval,Extruder\WObj:=Workobject_1;
MoveL RelTool (p1,65.500000,8.500000,9.428317,\Rx:=0.000000,\Ry:=11.442804),vel1,zoneval,Extruder\WObj:=Workobject_1;
MoveL RelTool (p1,63.000000,8.500000,11.921785,\Rx:=0.000000,\Ry:=8.251403),vel1,zoneval,Extruder\WObj:=Workobject_1;
MoveL RelTool (p1,60.500000,8.500000,13.556812,\Rx:=0.000000,\Ry:=5.898474),vel1,zoneval,Extruder\WObj:=Workobject_1;
MoveL RelTool (p1,58.000000,8.500000,14.736121,\Rx:=0.000000,\Ry:=4.733408),vel1,zoneval,Extruder\WObj:=Workobject_1;
MoveL RelTool (p1,55.500000,8.500000,15.637552,\Rx:=0.000000,\Ry:=3.655642),vel1,zoneval,Extruder\WObj:=Workobject_1;
MoveL RelTool (p1,53.000000,8.500000,16.339278,\Rx:=0.000000,\Ry:=2.815279),vel1,zoneval,Extruder\WObj:=Workobject_1;
MoveL RelTool (p1,50.500000,8.500000,16.851388,\Rx:=0.000000,\Ry:=1.924676),vel1,zoneval,Extruder\WObj:=Workobject_1;
MoveL RelTool (p1,48.000000,8.500000,17.213831,\Rx:=0.000000,\Ry:=1.178272),vel1,zoneval,Extruder\WObj:=Workobject_1;
MoveL RelTool (p1,45.500000,8.500000,17.425134,\Rx:=0.000000,\Ry:=0.578822),vel1,zoneval,Extruder\WObj:=Workobject_1;
MoveL RelTool (p1,43.000000,8.500000,17.491743,\Rx:=0.000000,\Ry:=0.047776),vel1,zoneval,Extruder\WObj:=Workobject_1;
MoveL RelTool (p1,40.500000,8.500000,17.421591,\Rx:=0.000000,\Ry:=-0.607859),vel1,zoneval,Extruder\WObj:=Workobject_1;
MoveL RelTool (p1,38.000000,8.500000,17.218209,\Rx:=0.000000,\Ry:=-1.457462),vel1,zoneval,Extruder\WObj:=Workobject_1;
MoveL RelTool (p1,35.500000,8.500000,16.878735,\Rx:=0.000000,\Ry:=-2.458274),vel1,zoneval,Extruder\WObj:=Workobject_1;
MoveL RelTool (p1,33.000000,8.500000,16.384292,\Rx:=0.000000,\Ry:=-3.167663),vel1,zoneval,Extruder\WObj:=Workobject_1;
MoveL RelTool (p1,30.500000,8.500000,15.704555,\Rx:=0.000000,\Ry:=-4.264941),vel1,zoneval,Extruder\WObj:=Workobject_1;
MoveL RelTool (p1,28.000000,8.500000,14.812629,\Rx:=0.000000,\Ry:=-5.359751),vel1,zoneval,Extruder\WObj:=Workobject_1;
MoveL RelTool (p1,25.500000,8.500000,13.636134,\Rx:=0.000000,\Ry:=-6.524894),vel1,zoneval,Extruder\WObj:=Workobject_1;
MoveL RelTool (p1,23.000000,8.500000,12.057248,\Rx:=0.000000,\Ry:=-8.365080),vel1,zoneval,Extruder\WObj:=Workobject_1;
MoveL RelTool (p1,20.500000,8.500000,9.659291,\Rx:=0.000000,\Ry:=-11.689062),vel1,zoneval,Extruder\WObj:=Workobject_1;
MoveL RelTool (p1,18.000000,8.500000,7.667393,\Rx:=0.000000,\Ry:=-2.952187),vel1,zoneval,Extruder\WObj:=Workobject_1;
MoveL RelTool (p1,15.500000,8.500000,7.500000,\Rx:=0.000000,\Ry:=0.000000),vel1,zoneval,Extruder\WObj:=Workobject_1;
MoveL RelTool (p1,13.000000,8.500000,7.500000,\Rx:=0.000000,\Ry:=0.000000),vel1,zoneval,Extruder\WObj:=Workobject_1;
MoveL RelTool (p1,10.500000,8.500000,7.500000,\Rx:=0.000000,\Ry:=0.000000),vel1,zoneval,Extruder\WObj:=Workobject_1;
MoveL RelTool (p1,8.000000,8.500000,7.500000,\Rx:=0.000000,\Ry:=0.000000),vel1,zoneval,Extruder\WObj:=Workobject_1;
MoveL RelTool (p1,5.500000,8.500000,7.500000,\Rx:=0.000000,\Ry:=0.000000),vel1,zoneval,Extruder\WObj:=Workobject_1;
MoveL RelTool (p1,3.000000,8.500000,7.500000,\Rx:=0.000000,\Ry:=0.000000),vel1,zoneval,Extruder\WObj:=Workobject_1;
MoveL RelTool (p1,5.000000,9.000000,7.500000,\Rx:=0.000000,\Ry:=-0.000000),vel1,zoneval,Extruder\WObj:=Workobject_1;
MoveL RelTool (p1,7.500000,9.000000,7.500000,\Rx:=0.000000,\Ry:=-0.000000),vel1,zoneval,Extruder\WObj:=Workobject_1;
MoveL RelTool (p1,10.000000,9.000000,7.500000,\Rx:=0.000000,\Ry:=-0.000000),vel1,zoneval,Extruder\WObj:=Workobject_1;
MoveL RelTool (p1,12.500000,9.000000,7.500000,\Rx:=0.000000,\Ry:=-0.000000),vel1,zoneval,Extruder\WObj:=Workobject_1;
MoveL RelTool (p1,15.000000,9.000000,7.500000,\Rx:=0.000000,\Ry:=-0.000000),vel1,zoneval,Extruder\WObj:=Workobject_1;
MoveL RelTool (p1,17.500000,9.000000,7.549338,\Rx:=0.000000,\Ry:=-2.952187),vel1,zoneval,Extruder\WObj:=Workobject_1;
MoveL RelTool (p1,20.000000,9.000000,9.005299,\Rx:=0.000000,\Ry:=-11.692806),vel1,zoneval,Extruder\WObj:=Workobject_1;
MoveL RelTool (p1,22.500000,9.000000,11.672110,\Rx:=0.000000,\Ry:=-8.376461),vel1,zoneval,Extruder\WObj:=Workobject_1;
MoveL RelTool (p1,25.000000,9.000000,13.355982,\Rx:=0.000000,\Ry:=-6.524894),vel1,zoneval,Extruder\WObj:=Workobject_1;
MoveL RelTool (p1,27.500000,9.000000,14.589646,\Rx:=0.000000,\Ry:=-5.360564),vel1,zoneval,Extruder\WObj:=Workobject_1;
MoveL RelTool (p1,30.000000,9.000000,15.530870,\Rx:=0.000000,\Ry:=-4.264941),vel1,zoneval,Extruder\WObj:=Workobject_1;
MoveL RelTool (p1,32.500000,9.000000,16.258326,\Rx:=0.000000,\Ry:=-3.139557),vel1,zoneval,Extruder\WObj:=Workobject_1;
MoveL RelTool (p1,35.000000,9.000000,16.781378,\Rx:=0.000000,\Ry:=-2.483640),vel1,zoneval,Extruder\WObj:=Workobject_1;
MoveL RelTool (p1,37.500000,9.000000,17.161388,\Rx:=0.000000,\Ry:=-1.457462),vel1,zoneval,Extruder\WObj:=Workobject_1;
MoveL RelTool (p1,40.000000,9.000000,17.398600,\Rx:=0.000000,\Ry:=-0.607859),vel1,zoneval,Extruder\WObj:=Workobject_1;
MoveL RelTool (p1,42.500000,9.000000,17.493505,\Rx:=0.000000,\Ry:=0.020090),vel1,zoneval,Extruder\WObj:=Workobject_1;
MoveL RelTool (p1,45.000000,9.000000,17.447698,\Rx:=0.000000,\Ry:=0.567557),vel1,zoneval,Extruder\WObj:=Workobject_1;
MoveL RelTool (p1,47.500000,9.000000,17.261058,\Rx:=0.000000,\Ry:=1.207076),vel1,zoneval,Extruder\WObj:=Workobject_1;
MoveL RelTool (p1,50.000000,9.000000,16.928029,\Rx:=0.000000,\Ry:=1.924676),vel1,zoneval,Extruder\WObj:=Workobject_1;
MoveL RelTool (p1,52.500000,9.000000,16.452652,\Rx:=0.000000,\Ry:=2.815279),vel1,zoneval,Extruder\WObj:=Workobject_1;
MoveL RelTool (p1,55.000000,9.000000,15.785206,\Rx:=0.000000,\Ry:=3.617426),vel1,zoneval,Extruder\WObj:=Workobject_1;
MoveL RelTool (p1,57.500000,9.000000,14.931773,\Rx:=0.000000,\Ry:=4.733408),vel1,zoneval,Extruder\WObj:=Workobject_1;
MoveL RelTool (p1,60.000000,9.000000,13.806864,\Rx:=0.000000,\Ry:=5.907601),vel1,zoneval,Extruder\WObj:=Workobject_1;
MoveL RelTool (p1,62.500000,9.000000,12.300679,\Rx:=0.000000,\Ry:=8.239916),vel1,zoneval,Extruder\WObj:=Workobject_1;
MoveL RelTool (p1,65.000000,9.000000,10.058244,\Rx:=0.000000,\Ry:=11.457668),vel1,zoneval,Extruder\WObj:=Workobject_1;
MoveL RelTool (p1,67.500000,9.000000,7.780757,\Rx:=0.000000,\Ry:=3.821551),vel1,zoneval,Extruder\WObj:=Workobject_1;
MoveL RelTool (p1,70.000000,9.000000,7.500000,\Rx:=0.000000,\Ry:=-0.000000),vel1,zoneval,Extruder\WObj:=Workobject_1;
MoveL RelTool (p1,72.500000,9.000000,7.500000,\Rx:=0.000000,\Ry:=-0.000000),vel1,zoneval,Extruder\WObj:=Workobject_1;
MoveL RelTool (p1,75.000000,9.000000,7.500000,\Rx:=0.000000,\Ry:=-0.000000),vel1,zoneval,Extruder\WObj:=Workobject_1;
MoveL RelTool (p1,77.500000,9.000000,7.500000,\Rx:=0.000000,\Ry:=-0.000000),vel1,zoneval,Extruder\WObj:=Workobject_1;
MoveL RelTool (p1,80.000000,9.000000,7.500000,\Rx:=0.000000,\Ry:=-0.000000),vel1,zoneval,Extruder\WObj:=Workobject_1;
MoveL RelTool (p1,82.500000,9.000000,7.500000,\Rx:=0.000000,\Ry:=-0.000000),vel1,zoneval,Extruder\WObj:=Workobject_1;
MoveL RelTool (p1,80.500000,9.500000,7.500000,\Rx:=0.000000,\Ry:=0.000000),vel1,zoneval,Extruder\WObj:=Workobject_1;
MoveL RelTool (p1,78.000000,9.500000,7.500000,\Rx:=0.000000,\Ry:=0.000000),vel1,zoneval,Extruder\WObj:=Workobject_1;
MoveL RelTool (p1,75.500000,9.500000,7.500000,\Rx:=0.000000,\Ry:=0.000000),vel1,zoneval,Extruder\WObj:=Workobject_1;
MoveL RelTool (p1,73.000000,9.500000,7.500000,\Rx:=0.000000,\Ry:=0.000000),vel1,zoneval,Extruder\WObj:=Workobject_1;
MoveL RelTool (p1,70.500000,9.500000,7.500000,\Rx:=0.000000,\Ry:=0.000000),vel1,zoneval,Extruder\WObj:=Workobject_1;
MoveL RelTool (p1,68.000000,9.500000,7.626010,\Rx:=0.000000,\Ry:=3.821551),vel1,zoneval,Extruder\WObj:=Workobject_1;
MoveL RelTool (p1,65.500000,9.500000,9.428317,\Rx:=0.000000,\Ry:=11.472488),vel1,zoneval,Extruder\WObj:=Workobject_1;
MoveL RelTool (p1,63.000000,9.500000,11.923839,\Rx:=0.000000,\Ry:=8.228414),vel1,zoneval,Extruder\WObj:=Workobject_1;
MoveL RelTool (p1,60.500000,9.500000,13.556499,\Rx:=0.000000,\Ry:=5.916722),vel1,zoneval,Extruder\WObj:=Workobject_1;
MoveL RelTool (p1,58.000000,9.500000,14.737535,\Rx:=0.000000,\Ry:=4.733408),vel1,zoneval,Extruder\WObj:=Workobject_1;
MoveL RelTool (p1,55.500000,9.500000,15.640849,\Rx:=0.000000,\Ry:=3.579142),vel1,zoneval,Extruder\WObj:=Workobject_1;
MoveL RelTool (p1,53.000000,9.500000,16.341239,\Rx:=0.000000,\Ry:=2.815279),vel1,zoneval,Extruder\WObj:=Workobject_1;
MoveL RelTool (p1,50.500000,9.500000,16.852344,\Rx:=0.000000,\Ry:=1.924676),vel1,zoneval,Extruder\WObj:=Workobject_1;
MoveL RelTool (p1,48.000000,9.500000,17.213196,\Rx:=0.000000,\Ry:=1.235868),vel1,zoneval,Extruder\WObj:=Workobject_1;
MoveL RelTool (p1,45.500000,9.500000,17.425658,\Rx:=0.000000,\Ry:=0.556291),vel1,zoneval,Extruder\WObj:=Workobject_1;
MoveL RelTool (p1,43.000000,9.500000,17.493012,\Rx:=0.000000,\Ry:=0.009614),vel1,zoneval,Extruder\WObj:=Workobject_1;
MoveL RelTool (p1,40.500000,9.500000,17.423387,\Rx:=0.000000,\Ry:=-0.607859),vel1,zoneval,Extruder\WObj:=Workobject_1;
MoveL RelTool (p1,38.000000,9.500000,17.219539,\Rx:=0.000000,\Ry:=-1.457462),vel1,zoneval,Extruder\WObj:=Workobject_1;
MoveL RelTool (p1,35.500000,9.500000,16.881598,\Rx:=0.000000,\Ry:=-2.483640),vel1,zoneval,Extruder\WObj:=Workobject_1;
MoveL RelTool (p1,33.000000,9.500000,16.384061,\Rx:=0.000000,\Ry:=-3.111420),vel1,zoneval,Extruder\WObj:=Workobject_1;
MoveL RelTool (p1,30.500000,9.500000,15.705269,\Rx:=0.000000,\Ry:=-4.264941),vel1,zoneval,Extruder\WObj:=Workobject_1;
MoveL RelTool (p1,28.000000,9.500000,14.814270,\Rx:=0.000000,\Ry:=-5.356618),vel1,zoneval,Extruder\WObj:=Workobject_1;
MoveL RelTool (p1,25.500000,9.500000,13.638428,\Rx:=0.000000,\Ry:=-6.524894),vel1,zoneval,Extruder\WObj:=Workobject_1;
MoveL RelTool (p1,23.000000,9.500000,12.059694,\Rx:=0.000000,\Ry:=-8.387826),vel1,zoneval,Extruder\WObj:=Workobject_1;
MoveL RelTool (p1,20.500000,9.500000,9.660088,\Rx:=0.000000,\Ry:=-11.696547),vel1,zoneval,Extruder\WObj:=Workobject_1;
MoveL RelTool (p1,18.000000,9.500000,7.667393,\Rx:=0.000000,\Ry:=-2.952187),vel1,zoneval,Extruder\WObj:=Workobject_1;
MoveL RelTool (p1,15.500000,9.500000,7.500000,\Rx:=0.000000,\Ry:=0.000000),vel1,zoneval,Extruder\WObj:=Workobject_1;
MoveL RelTool (p1,13.000000,9.500000,7.500000,\Rx:=0.000000,\Ry:=0.000000),vel1,zoneval,Extruder\WObj:=Workobject_1;
MoveL RelTool (p1,10.500000,9.500000,7.500000,\Rx:=0.000000,\Ry:=0.000000),vel1,zoneval,Extruder\WObj:=Workobject_1;
MoveL RelTool (p1,8.000000,9.500000,7.500000,\Rx:=0.000000,\Ry:=0.000000),vel1,zoneval,Extruder\WObj:=Workobject_1;
MoveL RelTool (p1,5.500000,9.500000,7.500000,\Rx:=0.000000,\Ry:=0.000000),vel1,zoneval,Extruder\WObj:=Workobject_1;
MoveL RelTool (p1,3.000000,9.500000,7.500000,\Rx:=0.000000,\Ry:=0.000000),vel1,zoneval,Extruder\WObj:=Workobject_1;
MoveL RelTool (p1,5.000000,10.000000,7.500000,\Rx:=0.000000,\Ry:=-0.000000),vel1,zoneval,Extruder\WObj:=Workobject_1;
MoveL RelTool (p1,7.500000,10.000000,7.500000,\Rx:=0.000000,\Ry:=-0.000000),vel1,zoneval,Extruder\WObj:=Workobject_1;
MoveL RelTool (p1,10.000000,10.000000,7.500000,\Rx:=0.000000,\Ry:=-0.000000),vel1,zoneval,Extruder\WObj:=Workobject_1;
MoveL RelTool (p1,12.500000,10.000000,7.500000,\Rx:=0.000000,\Ry:=-0.000000),vel1,zoneval,Extruder\WObj:=Workobject_1;
MoveL RelTool (p1,15.000000,10.000000,7.500000,\Rx:=0.000000,\Ry:=-0.000000),vel1,zoneval,Extruder\WObj:=Workobject_1;
MoveL RelTool (p1,17.500000,10.000000,7.549338,\Rx:=0.000000,\Ry:=-2.952187),vel1,zoneval,Extruder\WObj:=Workobject_1;
MoveL RelTool (p1,20.000000,10.000000,9.005299,\Rx:=0.000000,\Ry:=-11.700285),vel1,zoneval,Extruder\WObj:=Workobject_1;
MoveL RelTool (p1,22.500000,10.000000,11.673130,\Rx:=0.000000,\Ry:=-8.399175),vel1,zoneval,Extruder\WObj:=Workobject_1;
MoveL RelTool (p1,25.000000,10.000000,13.358277,\Rx:=0.000000,\Ry:=-6.524894),vel1,zoneval,Extruder\WObj:=Workobject_1;
MoveL RelTool (p1,27.500000,10.000000,14.591472,\Rx:=0.000000,\Ry:=-5.330022),vel1,zoneval,Extruder\WObj:=Workobject_1;
MoveL RelTool (p1,30.000000,10.000000,15.531583,\Rx:=0.000000,\Ry:=-4.264941),vel1,zoneval,Extruder\WObj:=Workobject_1;
MoveL RelTool (p1,32.500000,10.000000,16.260443,\Rx:=0.000000,\Ry:=-3.083252),vel1,zoneval,Extruder\WObj:=Workobject_1;
MoveL RelTool (p1,35.000000,10.000000,16.784241,\Rx:=0.000000,\Ry:=-2.483640),vel1,zoneval,Extruder\WObj:=Workobject_1;
MoveL RelTool (p1,37.500000,10.000000,17.162718,\Rx:=0.000000,\Ry:=-1.457462),vel1,zoneval,Extruder\WObj:=Workobject_1;
MoveL RelTool (p1,40.000000,10.000000,17.400396,\Rx:=0.000000,\Ry:=-0.607859),vel1,zoneval,Extruder\WObj:=Workobject_1;
MoveL RelTool (p1,42.500000,10.000000,17.493275,\Rx:=0.000000,\Ry:=0.009614),vel1,zoneval,Extruder\WObj:=Workobject_1;
MoveL RelTool (p1,45.000000,10.000000,17.447336,\Rx:=0.000000,\Ry:=0.545025),vel1,zoneval,Extruder\WObj:=Workobject_1;
MoveL RelTool (p1,47.500000,10.000000,17.262705,\Rx:=0.000000,\Ry:=1.264647),vel1,zoneval,Extruder\WObj:=Workobject_1;
MoveL RelTool (p1,50.000000,10.000000,16.928984,\Rx:=0.000000,\Ry:=1.924676),vel1,zoneval,Extruder\WObj:=Workobject_1;
MoveL RelTool (p1,52.500000,10.000000,16.454613,\Rx:=0.000000,\Ry:=2.817973),vel1,zoneval,Extruder\WObj:=Workobject_1;
MoveL RelTool (p1,55.000000,10.000000,15.786013,\Rx:=0.000000,\Ry:=3.558921),vel1,zoneval,Extruder\WObj:=Workobject_1;
MoveL RelTool (p1,57.500000,10.000000,14.933187,\Rx:=0.000000,\Ry:=4.733408),vel1,zoneval,Extruder\WObj:=Workobject_1;
MoveL RelTool (p1,60.000000,10.000000,13.807447,\Rx:=0.000000,\Ry:=5.925836),vel1,zoneval,Extruder\WObj:=Workobject_1;
MoveL RelTool (p1,62.500000,10.000000,12.301315,\Rx:=0.000000,\Ry:=8.216896),vel1,zoneval,Extruder\WObj:=Workobject_1;
MoveL RelTool (p1,65.000000,10.000000,10.061260,\Rx:=0.000000,\Ry:=11.487265),vel1,zoneval,Extruder\WObj:=Workobject_1;
MoveL RelTool (p1,67.500000,10.000000,7.780757,\Rx:=0.000000,\Ry:=3.821551),vel1,zoneval,Extruder\WObj:=Workobject_1;
MoveL RelTool (p1,70.000000,10.000000,7.500000,\Rx:=0.000000,\Ry:=-0.000000),vel1,zoneval,Extruder\WObj:=Workobject_1;
MoveL RelTool (p1,72.500000,10.000000,7.500000,\Rx:=0.000000,\Ry:=-0.000000),vel1,zoneval,Extruder\WObj:=Workobject_1;
MoveL RelTool (p1,75.000000,10.000000,7.500000,\Rx:=0.000000,\Ry:=-0.000000),vel1,zoneval,Extruder\WObj:=Workobject_1;
MoveL RelTool (p1,77.500000,10.000000,7.500000,\Rx:=0.000000,\Ry:=-0.000000),vel1,zoneval,Extruder\WObj:=Workobject_1;
MoveL RelTool (p1,80.000000,10.000000,7.500000,\Rx:=0.000000,\Ry:=-0.000000),vel1,zoneval,Extruder\WObj:=Workobject_1;
MoveL RelTool (p1,82.500000,10.000000,7.500000,\Rx:=0.000000,\Ry:=-0.000000),vel1,zoneval,Extruder\WObj:=Workobject_1;
MoveL RelTool (p1,80.500000,10.500000,7.500000,\Rx:=0.000000,\Ry:=0.000000),vel1,zoneval,Extruder\WObj:=Workobject_1;
MoveL RelTool (p1,78.000000,10.500000,7.500000,\Rx:=0.000000,\Ry:=0.000000),vel1,zoneval,Extruder\WObj:=Workobject_1;
MoveL RelTool (p1,75.500000,10.500000,7.500000,\Rx:=0.000000,\Ry:=0.000000),vel1,zoneval,Extruder\WObj:=Workobject_1;
MoveL RelTool (p1,73.000000,10.500000,7.500000,\Rx:=0.000000,\Ry:=0.000000),vel1,zoneval,Extruder\WObj:=Workobject_1;
MoveL RelTool (p1,70.500000,10.500000,7.500000,\Rx:=0.000000,\Ry:=0.000000),vel1,zoneval,Extruder\WObj:=Workobject_1;
MoveL RelTool (p1,68.000000,10.500000,7.626010,\Rx:=0.000000,\Ry:=3.821551),vel1,zoneval,Extruder\WObj:=Workobject_1;
MoveL RelTool (p1,65.500000,10.500000,9.428317,\Rx:=0.000000,\Ry:=11.501998),vel1,zoneval,Extruder\WObj:=Workobject_1;
MoveL RelTool (p1,63.000000,10.500000,11.925892,\Rx:=0.000000,\Ry:=8.205362),vel1,zoneval,Extruder\WObj:=Workobject_1;
MoveL RelTool (p1,60.500000,10.500000,13.556185,\Rx:=0.000000,\Ry:=5.934943),vel1,zoneval,Extruder\WObj:=Workobject_1;
MoveL RelTool (p1,58.000000,10.500000,14.738948,\Rx:=0.000000,\Ry:=4.733408),vel1,zoneval,Extruder\WObj:=Workobject_1;
MoveL RelTool (p1,55.500000,10.500000,15.644145,\Rx:=0.000000,\Ry:=3.558921),vel1,zoneval,Extruder\WObj:=Workobject_1;
MoveL RelTool (p1,53.000000,10.500000,16.342126,\Rx:=0.000000,\Ry:=2.841296),vel1,zoneval,Extruder\WObj:=Workobject_1;
MoveL RelTool (p1,50.500000,10.500000,16.853299,\Rx:=0.000000,\Ry:=1.924676),vel1,zoneval,Extruder\WObj:=Workobject_1;
MoveL RelTool (p1,48.000000,10.500000,17.212561,\Rx:=0.000000,\Ry:=1.293414),vel1,zoneval,Extruder\WObj:=Workobject_1;
MoveL RelTool (p1,45.500000,10.500000,17.426182,\Rx:=0.000000,\Ry:=0.533757),vel1,zoneval,Extruder\WObj:=Workobject_1;
MoveL RelTool (p1,43.000000,10.500000,17.492783,\Rx:=0.000000,\Ry:=0.009614),vel1,zoneval,Extruder\WObj:=Workobject_1;
MoveL RelTool (p1,40.500000,10.500000,17.425183,\Rx:=0.000000,\Ry:=-0.607859),vel1,zoneval,Extruder\WObj:=Workobject_1;
MoveL RelTool (p1,38.000000,10.500000,17.220869,\Rx:=0.000000,\Ry:=-1.457981),vel1,zoneval,Extruder\WObj:=Workobject_1;
MoveL RelTool (p1,35.500000,10.500000,16.884461,\Rx:=0.000000,\Ry:=-2.483640),vel1,zoneval,Extruder\WObj:=Workobject_1;
MoveL RelTool (p1,33.000000,10.500000,16.383830,\Rx:=0.000000,\Ry:=-3.055053),vel1,zoneval,Extruder\WObj:=Workobject_1;
MoveL RelTool (p1,30.500000,10.500000,15.705982,\Rx:=0.000000,\Ry:=-4.264941),vel1,zoneval,Extruder\WObj:=Workobject_1;
MoveL RelTool (p1,28.000000,10.500000,14.813592,\Rx:=0.000000,\Ry:=-5.303377),vel1,zoneval,Extruder\WObj:=Workobject_1;
MoveL RelTool (p1,25.500000,10.500000,13.640723,\Rx:=0.000000,\Ry:=-6.524894),vel1,zoneval,Extruder\WObj:=Workobject_1;
MoveL RelTool (p1,23.000000,10.500000,12.060783,\Rx:=0.000000,\Ry:=-8.388916),vel1,zoneval,Extruder\WObj:=Workobject_1;
MoveL RelTool (p1,20.500000,10.500000,9.660886,\Rx:=0.000000,\Ry:=-11.704021),vel1,zoneval,Extruder\WObj:=Workobject_1;
MoveL RelTool (p1,18.000000,10.500000,7.667393,\Rx:=0.000000,\Ry:=-2.952187),vel1,zoneval,Extruder\WObj:=Workobject_1;
MoveL RelTool (p1,15.500000,10.500000,7.500000,\Rx:=0.000000,\Ry:=0.000000),vel1,zoneval,Extruder\WObj:=Workobject_1;
MoveL RelTool (p1,13.000000,10.500000,7.500000,\Rx:=0.000000,\Ry:=0.000000),vel1,zoneval,Extruder\WObj:=Workobject_1;
MoveL RelTool (p1,10.500000,10.500000,7.500000,\Rx:=0.000000,\Ry:=0.000000),vel1,zoneval,Extruder\WObj:=Workobject_1;
MoveL RelTool (p1,8.000000,10.500000,7.500000,\Rx:=0.000000,\Ry:=0.000000),vel1,zoneval,Extruder\WObj:=Workobject_1;
MoveL RelTool (p1,5.500000,10.500000,7.500000,\Rx:=0.000000,\Ry:=0.000000),vel1,zoneval,Extruder\WObj:=Workobject_1;
MoveL RelTool (p1,3.000000,10.500000,7.500000,\Rx:=0.000000,\Ry:=0.000000),vel1,zoneval,Extruder\WObj:=Workobject_1;
MoveL RelTool (p1,5.000000,11.000000,7.500000,\Rx:=0.000000,\Ry:=-0.000000),vel1,zoneval,Extruder\WObj:=Workobject_1;
MoveL RelTool (p1,7.500000,11.000000,7.500000,\Rx:=0.000000,\Ry:=-0.000000),vel1,zoneval,Extruder\WObj:=Workobject_1;
MoveL RelTool (p1,10.000000,11.000000,7.500000,\Rx:=0.000000,\Ry:=-0.000000),vel1,zoneval,Extruder\WObj:=Workobject_1;
MoveL RelTool (p1,12.500000,11.000000,7.500000,\Rx:=0.000000,\Ry:=-0.000000),vel1,zoneval,Extruder\WObj:=Workobject_1;
MoveL RelTool (p1,15.000000,11.000000,7.500000,\Rx:=0.000000,\Ry:=-0.000000),vel1,zoneval,Extruder\WObj:=Workobject_1;
MoveL RelTool (p1,17.500000,11.000000,7.549338,\Rx:=0.000000,\Ry:=-2.952187),vel1,zoneval,Extruder\WObj:=Workobject_1;
MoveL RelTool (p1,20.000000,11.000000,9.005299,\Rx:=0.000000,\Ry:=-11.707753),vel1,zoneval,Extruder\WObj:=Workobject_1;
MoveL RelTool (p1,22.500000,11.000000,11.674150,\Rx:=0.000000,\Ry:=-8.377137),vel1,zoneval,Extruder\WObj:=Workobject_1;
MoveL RelTool (p1,25.000000,11.000000,13.360572,\Rx:=0.000000,\Ry:=-6.524894),vel1,zoneval,Extruder\WObj:=Workobject_1;
MoveL RelTool (p1,27.500000,11.000000,14.593299,\Rx:=0.000000,\Ry:=-5.276683),vel1,zoneval,Extruder\WObj:=Workobject_1;
MoveL RelTool (p1,30.000000,11.000000,15.532296,\Rx:=0.000000,\Ry:=-4.264941),vel1,zoneval,Extruder\WObj:=Workobject_1;
MoveL RelTool (p1,32.500000,11.000000,16.262561,\Rx:=0.000000,\Ry:=-3.026823),vel1,zoneval,Extruder\WObj:=Workobject_1;
MoveL RelTool (p1,35.000000,11.000000,16.787104,\Rx:=0.000000,\Ry:=-2.483640),vel1,zoneval,Extruder\WObj:=Workobject_1;
MoveL RelTool (p1,37.500000,11.000000,17.164004,\Rx:=0.000000,\Ry:=-1.458589),vel1,zoneval,Extruder\WObj:=Workobject_1;
MoveL RelTool (p1,40.000000,11.000000,17.402192,\Rx:=0.000000,\Ry:=-0.607859),vel1,zoneval,Extruder\WObj:=Workobject_1;
MoveL RelTool (p1,42.500000,11.000000,17.493046,\Rx:=0.000000,\Ry:=0.009614),vel1,zoneval,Extruder\WObj:=Workobject_1;
MoveL RelTool (p1,45.000000,11.000000,17.446973,\Rx:=0.000000,\Ry:=0.522489),vel1,zoneval,Extruder\WObj:=Workobject_1;
MoveL RelTool (p1,47.500000,11.000000,17.264352,\Rx:=0.000000,\Ry:=1.322167),vel1,zoneval,Extruder\WObj:=Workobject_1;
MoveL RelTool (p1,50.000000,11.000000,16.929939,\Rx:=0.000000,\Ry:=1.924676),vel1,zoneval,Extruder\WObj:=Workobject_1;
MoveL RelTool (p1,52.500000,11.000000,16.456574,\Rx:=0.000000,\Ry:=2.864600),vel1,zoneval,Extruder\WObj:=Workobject_1;
MoveL RelTool (p1,55.000000,11.000000,15.789309,\Rx:=0.000000,\Ry:=3.558921),vel1,zoneval,Extruder\WObj:=Workobject_1;
MoveL RelTool (p1,57.500000,11.000000,14.934601,\Rx:=0.000000,\Ry:=4.733408),vel1,zoneval,Extruder\WObj:=Workobject_1;
MoveL RelTool (p1,60.000000,11.000000,13.808030,\Rx:=0.000000,\Ry:=5.944044),vel1,zoneval,Extruder\WObj:=Workobject_1;
MoveL RelTool (p1,62.500000,11.000000,12.301950,\Rx:=0.000000,\Ry:=8.193812),vel1,zoneval,Extruder\WObj:=Workobject_1;
MoveL RelTool (p1,65.000000,11.000000,10.063527,\Rx:=0.000000,\Ry:=11.509397),vel1,zoneval,Extruder\WObj:=Workobject_1;
MoveL RelTool (p1,67.500000,11.000000,7.780757,\Rx:=0.000000,\Ry:=3.821551),vel1,zoneval,Extruder\WObj:=Workobject_1;
MoveL RelTool (p1,70.000000,11.000000,7.500000,\Rx:=0.000000,\Ry:=-0.000000),vel1,zoneval,Extruder\WObj:=Workobject_1;
MoveL RelTool (p1,72.500000,11.000000,7.500000,\Rx:=0.000000,\Ry:=-0.000000),vel1,zoneval,Extruder\WObj:=Workobject_1;
MoveL RelTool (p1,75.000000,11.000000,7.500000,\Rx:=0.000000,\Ry:=-0.000000),vel1,zoneval,Extruder\WObj:=Workobject_1;
MoveL RelTool (p1,77.500000,11.000000,7.500000,\Rx:=0.000000,\Ry:=-0.000000),vel1,zoneval,Extruder\WObj:=Workobject_1;
MoveL RelTool (p1,80.000000,11.000000,7.500000,\Rx:=0.000000,\Ry:=-0.000000),vel1,zoneval,Extruder\WObj:=Workobject_1;
MoveL RelTool (p1,82.500000,11.000000,7.500000,\Rx:=0.000000,\Ry:=-0.000000),vel1,zoneval,Extruder\WObj:=Workobject_1;
MoveL RelTool (p1,80.500000,11.500000,7.500000,\Rx:=0.000000,\Ry:=0.000000),vel1,zoneval,Extruder\WObj:=Workobject_1;
MoveL RelTool (p1,78.000000,11.500000,7.500000,\Rx:=0.000000,\Ry:=0.000000),vel1,zoneval,Extruder\WObj:=Workobject_1;
MoveL RelTool (p1,75.500000,11.500000,7.500000,\Rx:=0.000000,\Ry:=0.000000),vel1,zoneval,Extruder\WObj:=Workobject_1;
MoveL RelTool (p1,73.000000,11.500000,7.500000,\Rx:=0.000000,\Ry:=0.000000),vel1,zoneval,Extruder\WObj:=Workobject_1;
MoveL RelTool (p1,70.500000,11.500000,7.500000,\Rx:=0.000000,\Ry:=0.000000),vel1,zoneval,Extruder\WObj:=Workobject_1;
MoveL RelTool (p1,68.000000,11.500000,7.626010,\Rx:=0.000000,\Ry:=3.821551),vel1,zoneval,Extruder\WObj:=Workobject_1;
MoveL RelTool (p1,65.500000,11.500000,9.428317,\Rx:=0.000000,\Ry:=11.505970),vel1,zoneval,Extruder\WObj:=Workobject_1;
MoveL RelTool (p1,63.000000,11.500000,11.927946,\Rx:=0.000000,\Ry:=8.182247),vel1,zoneval,Extruder\WObj:=Workobject_1;
MoveL RelTool (p1,60.500000,11.500000,13.555872,\Rx:=0.000000,\Ry:=5.953139),vel1,zoneval,Extruder\WObj:=Workobject_1;
MoveL RelTool (p1,58.000000,11.500000,14.740362,\Rx:=0.000000,\Ry:=4.733408),vel1,zoneval,Extruder\WObj:=Workobject_1;
MoveL RelTool (p1,55.500000,11.500000,15.647442,\Rx:=0.000000,\Ry:=3.558921),vel1,zoneval,Extruder\WObj:=Workobject_1;
MoveL RelTool (p1,53.000000,11.500000,16.342162,\Rx:=0.000000,\Ry:=2.887884),vel1,zoneval,Extruder\WObj:=Workobject_1;
MoveL RelTool (p1,50.500000,11.500000,16.854254,\Rx:=0.000000,\Ry:=1.924676),vel1,zoneval,Extruder\WObj:=Workobject_1;
MoveL RelTool (p1,48.000000,11.500000,17.211926,\Rx:=0.000000,\Ry:=1.350906),vel1,zoneval,Extruder\WObj:=Workobject_1;
MoveL RelTool (p1,45.500000,11.500000,17.426706,\Rx:=0.000000,\Ry:=0.511220),vel1,zoneval,Extruder\WObj:=Workobject_1;
MoveL RelTool (p1,43.000000,11.500000,17.492554,\Rx:=0.000000,\Ry:=0.009614),vel1,zoneval,Extruder\WObj:=Workobject_1;
MoveL RelTool (p1,40.500000,11.500000,17.426978,\Rx:=0.000000,\Ry:=-0.607859),vel1,zoneval,Extruder\WObj:=Workobject_1;
MoveL RelTool (p1,38.000000,11.500000,17.222199,\Rx:=0.000000,\Ry:=-1.459197),vel1,zoneval,Extruder\WObj:=Workobject_1;
MoveL RelTool (p1,35.500000,11.500000,16.887324,\Rx:=0.000000,\Ry:=-2.483640),vel1,zoneval,Extruder\WObj:=Workobject_1;
MoveL RelTool (p1,33.000000,11.500000,16.383599,\Rx:=0.000000,\Ry:=-3.021941),vel1,zoneval,Extruder\WObj:=Workobject_1;
MoveL RelTool (p1,30.500000,11.500000,15.706695,\Rx:=0.000000,\Ry:=-4.264941),vel1,zoneval,Extruder\WObj:=Workobject_1;
MoveL RelTool (p1,28.000000,11.500000,14.812914,\Rx:=0.000000,\Ry:=-5.249939),vel1,zoneval,Extruder\WObj:=Workobject_1;
MoveL RelTool (p1,25.500000,11.500000,13.643018,\Rx:=0.000000,\Ry:=-6.524894),vel1,zoneval,Extruder\WObj:=Workobject_1;
MoveL RelTool (p1,23.000000,11.500000,12.060324,\Rx:=0.000000,\Ry:=-8.365341),vel1,zoneval,Extruder\WObj:=Workobject_1;
MoveL RelTool (p1,20.500000,11.500000,9.661683,\Rx:=0.000000,\Ry:=-11.711483),vel1,zoneval,Extruder\WObj:=Workobject_1;
MoveL RelTool (p1,18.000000,11.500000,7.667393,\Rx:=0.000000,\Ry:=-2.952187),vel1,zoneval,Extruder\WObj:=Workobject_1;
MoveL RelTool (p1,15.500000,11.500000,7.500000,\Rx:=0.000000,\Ry:=0.000000),vel1,zoneval,Extruder\WObj:=Workobject_1;
MoveL RelTool (p1,13.000000,11.500000,7.500000,\Rx:=0.000000,\Ry:=0.000000),vel1,zoneval,Extruder\WObj:=Workobject_1;
MoveL RelTool (p1,10.500000,11.500000,7.500000,\Rx:=0.000000,\Ry:=0.000000),vel1,zoneval,Extruder\WObj:=Workobject_1;
MoveL RelTool (p1,8.000000,11.500000,7.500000,\Rx:=0.000000,\Ry:=0.000000),vel1,zoneval,Extruder\WObj:=Workobject_1;
MoveL RelTool (p1,5.500000,11.500000,7.500000,\Rx:=0.000000,\Ry:=0.000000),vel1,zoneval,Extruder\WObj:=Workobject_1;
MoveL RelTool (p1,3.000000,11.500000,7.500000,\Rx:=0.000000,\Ry:=0.000000),vel1,zoneval,Extruder\WObj:=Workobject_1;
MoveL RelTool (p1,5.000000,12.000000,7.500000,\Rx:=0.000000,\Ry:=-0.000000),vel1,zoneval,Extruder\WObj:=Workobject_1;
MoveL RelTool (p1,7.500000,12.000000,7.500000,\Rx:=0.000000,\Ry:=-0.000000),vel1,zoneval,Extruder\WObj:=Workobject_1;
MoveL RelTool (p1,10.000000,12.000000,7.500000,\Rx:=0.000000,\Ry:=-0.000000),vel1,zoneval,Extruder\WObj:=Workobject_1;
MoveL RelTool (p1,12.500000,12.000000,7.500000,\Rx:=0.000000,\Ry:=-0.000000),vel1,zoneval,Extruder\WObj:=Workobject_1;
MoveL RelTool (p1,15.000000,12.000000,7.500000,\Rx:=0.000000,\Ry:=-0.000000),vel1,zoneval,Extruder\WObj:=Workobject_1;
MoveL RelTool (p1,17.500000,12.000000,7.549338,\Rx:=0.000000,\Ry:=-2.952187),vel1,zoneval,Extruder\WObj:=Workobject_1;
MoveL RelTool (p1,20.000000,12.000000,9.005299,\Rx:=0.000000,\Ry:=-11.715209),vel1,zoneval,Extruder\WObj:=Workobject_1;
MoveL RelTool (p1,22.500000,12.000000,11.675169,\Rx:=0.000000,\Ry:=-8.353529),vel1,zoneval,Extruder\WObj:=Workobject_1;
MoveL RelTool (p1,25.000000,12.000000,13.362866,\Rx:=0.000000,\Ry:=-6.524894),vel1,zoneval,Extruder\WObj:=Workobject_1;
MoveL RelTool (p1,27.500000,12.000000,14.595126,\Rx:=0.000000,\Ry:=-5.223146),vel1,zoneval,Extruder\WObj:=Workobject_1;
MoveL RelTool (p1,30.000000,12.000000,15.533010,\Rx:=0.000000,\Ry:=-4.264941),vel1,zoneval,Extruder\WObj:=Workobject_1;
MoveL RelTool (p1,32.500000,12.000000,16.262533,\Rx:=0.000000,\Ry:=-3.021941),vel1,zoneval,Extruder\WObj:=Workobject_1;
MoveL RelTool (p1,35.000000,12.000000,16.789967,\Rx:=0.000000,\Ry:=-2.471187),vel1,zoneval,Extruder\WObj:=Workobject_1;
MoveL RelTool (p1,37.500000,12.000000,17.165286,\Rx:=0.000000,\Ry:=-1.459805),vel1,zoneval,Extruder\WObj:=Workobject_1;
MoveL RelTool (p1,40.000000,12.000000,17.403988,\Rx:=0.000000,\Ry:=-0.607859),vel1,zoneval,Extruder\WObj:=Workobject_1;
MoveL RelTool (p1,42.500000,12.000000,17.492817,\Rx:=0.000000,\Ry:=0.009614),vel1,zoneval,Extruder\WObj:=Workobject_1;
MoveL RelTool (p1,45.000000,12.000000,17.446611,\Rx:=0.000000,\Ry:=0.499950),vel1,zoneval,Extruder\WObj:=Workobject_1;
MoveL RelTool (p1,47.500000,12.000000,17.265999,\Rx:=0.000000,\Ry:=1.379632),vel1,zoneval,Extruder\WObj:=Workobject_1;
MoveL RelTool (p1,50.000000,12.000000,16.930894,\Rx:=0.000000,\Ry:=1.924676),vel1,zoneval,Extruder\WObj:=Workobject_1;
MoveL RelTool (p1,52.500000,12.000000,16.458535,\Rx:=0.000000,\Ry:=2.911149),vel1,zoneval,Extruder\WObj:=Workobject_1;
MoveL RelTool (p1,55.000000,12.000000,15.792606,\Rx:=0.000000,\Ry:=3.558921),vel1,zoneval,Extruder\WObj:=Workobject_1;
MoveL RelTool (p1,57.500000,12.000000,14.936009,\Rx:=0.000000,\Ry:=4.733289),vel1,zoneval,Extruder\WObj:=Workobject_1;
MoveL RelTool (p1,60.000000,12.000000,13.808612,\Rx:=0.000000,\Ry:=5.962227),vel1,zoneval,Extruder\WObj:=Workobject_1;
MoveL RelTool (p1,62.500000,12.000000,12.302585,\Rx:=0.000000,\Ry:=8.170666),vel1,zoneval,Extruder\WObj:=Workobject_1;
MoveL RelTool (p1,65.000000,12.000000,10.062824,\Rx:=0.000000,\Ry:=11.502541),vel1,zoneval,Extruder\WObj:=Workobject_1;
MoveL RelTool (p1,67.500000,12.000000,7.780757,\Rx:=0.000000,\Ry:=3.821551),vel1,zoneval,Extruder\WObj:=Workobject_1;
MoveL RelTool (p1,70.000000,12.000000,7.500000,\Rx:=0.000000,\Ry:=-0.000000),vel1,zoneval,Extruder\WObj:=Workobject_1;
MoveL RelTool (p1,72.500000,12.000000,7.500000,\Rx:=0.000000,\Ry:=-0.000000),vel1,zoneval,Extruder\WObj:=Workobject_1;
MoveL RelTool (p1,75.000000,12.000000,7.500000,\Rx:=0.000000,\Ry:=-0.000000),vel1,zoneval,Extruder\WObj:=Workobject_1;
MoveL RelTool (p1,77.500000,12.000000,7.500000,\Rx:=0.000000,\Ry:=-0.000000),vel1,zoneval,Extruder\WObj:=Workobject_1;
MoveL RelTool (p1,80.000000,12.000000,7.500000,\Rx:=0.000000,\Ry:=-0.000000),vel1,zoneval,Extruder\WObj:=Workobject_1;
MoveL RelTool (p1,82.500000,12.000000,7.500000,\Rx:=0.000000,\Ry:=-0.000000),vel1,zoneval,Extruder\WObj:=Workobject_1;
MoveL RelTool (p1,80.500000,12.500000,7.500000,\Rx:=0.000000,\Ry:=0.000000),vel1,zoneval,Extruder\WObj:=Workobject_1;
MoveL RelTool (p1,78.000000,12.500000,7.500000,\Rx:=0.000000,\Ry:=0.000000),vel1,zoneval,Extruder\WObj:=Workobject_1;
MoveL RelTool (p1,75.500000,12.500000,7.500000,\Rx:=0.000000,\Ry:=0.000000),vel1,zoneval,Extruder\WObj:=Workobject_1;
MoveL RelTool (p1,73.000000,12.500000,7.500000,\Rx:=0.000000,\Ry:=0.000000),vel1,zoneval,Extruder\WObj:=Workobject_1;
MoveL RelTool (p1,70.500000,12.500000,7.500000,\Rx:=0.000000,\Ry:=0.000000),vel1,zoneval,Extruder\WObj:=Workobject_1;
MoveL RelTool (p1,68.000000,12.500000,7.626010,\Rx:=0.000000,\Ry:=3.821551),vel1,zoneval,Extruder\WObj:=Workobject_1;
MoveL RelTool (p1,65.500000,12.500000,9.428317,\Rx:=0.000000,\Ry:=11.499110),vel1,zoneval,Extruder\WObj:=Workobject_1;
MoveL RelTool (p1,63.000000,12.500000,11.929999,\Rx:=0.000000,\Ry:=8.159069),vel1,zoneval,Extruder\WObj:=Workobject_1;
MoveL RelTool (p1,60.500000,12.500000,13.555559,\Rx:=0.000000,\Ry:=5.971308),vel1,zoneval,Extruder\WObj:=Workobject_1;
MoveL RelTool (p1,58.000000,12.500000,14.741776,\Rx:=0.000000,\Ry:=4.728908),vel1,zoneval,Extruder\WObj:=Workobject_1;
MoveL RelTool (p1,55.500000,12.500000,15.650738,\Rx:=0.000000,\Ry:=3.558921),vel1,zoneval,Extruder\WObj:=Workobject_1;
MoveL RelTool (p1,53.000000,12.500000,16.342198,\Rx:=0.000000,\Ry:=2.934394),vel1,zoneval,Extruder\WObj:=Workobject_1;
MoveL RelTool (p1,50.500000,12.500000,16.855209,\Rx:=0.000000,\Ry:=1.929388),vel1,zoneval,Extruder\WObj:=Workobject_1;
MoveL RelTool (p1,48.000000,12.500000,17.211291,\Rx:=0.000000,\Ry:=1.408344),vel1,zoneval,Extruder\WObj:=Workobject_1;
MoveL RelTool (p1,45.500000,12.500000,17.426866,\Rx:=0.000000,\Ry:=0.497915),vel1,zoneval,Extruder\WObj:=Workobject_1;
MoveL RelTool (p1,43.000000,12.500000,17.492324,\Rx:=0.000000,\Ry:=0.009614),vel1,zoneval,Extruder\WObj:=Workobject_1;
MoveL RelTool (p1,40.500000,12.500000,17.428774,\Rx:=0.000000,\Ry:=-0.618872),vel1,zoneval,Extruder\WObj:=Workobject_1;
MoveL RelTool (p1,38.000000,12.500000,17.223530,\Rx:=0.000000,\Ry:=-1.460413),vel1,zoneval,Extruder\WObj:=Workobject_1;
MoveL RelTool (p1,35.500000,12.500000,16.887943,\Rx:=0.000000,\Ry:=-2.428595),vel1,zoneval,Extruder\WObj:=Workobject_1;
MoveL RelTool (p1,33.000000,12.500000,16.383369,\Rx:=0.000000,\Ry:=-3.021941),vel1,zoneval,Extruder\WObj:=Workobject_1;
MoveL RelTool (p1,30.500000,12.500000,15.707409,\Rx:=0.000000,\Ry:=-4.264941),vel1,zoneval,Extruder\WObj:=Workobject_1;
MoveL RelTool (p1,28.000000,12.500000,14.812236,\Rx:=0.000000,\Ry:=-5.196304),vel1,zoneval,Extruder\WObj:=Workobject_1;
MoveL RelTool (p1,25.500000,12.500000,13.645313,\Rx:=0.000000,\Ry:=-6.530409),vel1,zoneval,Extruder\WObj:=Workobject_1;
MoveL RelTool (p1,23.000000,12.500000,12.059865,\Rx:=0.000000,\Ry:=-8.341700),vel1,zoneval,Extruder\WObj:=Workobject_1;
MoveL RelTool (p1,20.500000,12.500000,9.662480,\Rx:=0.000000,\Ry:=-11.718933),vel1,zoneval,Extruder\WObj:=Workobject_1;
MoveL RelTool (p1,18.000000,12.500000,7.667393,\Rx:=0.000000,\Ry:=-2.952187),vel1,zoneval,Extruder\WObj:=Workobject_1;
MoveL RelTool (p1,15.500000,12.500000,7.500000,\Rx:=0.000000,\Ry:=0.000000),vel1,zoneval,Extruder\WObj:=Workobject_1;
MoveL RelTool (p1,13.000000,12.500000,7.500000,\Rx:=0.000000,\Ry:=0.000000),vel1,zoneval,Extruder\WObj:=Workobject_1;
MoveL RelTool (p1,10.500000,12.500000,7.500000,\Rx:=0.000000,\Ry:=0.000000),vel1,zoneval,Extruder\WObj:=Workobject_1;
MoveL RelTool (p1,8.000000,12.500000,7.500000,\Rx:=0.000000,\Ry:=0.000000),vel1,zoneval,Extruder\WObj:=Workobject_1;
MoveL RelTool (p1,5.500000,12.500000,7.500000,\Rx:=0.000000,\Ry:=0.000000),vel1,zoneval,Extruder\WObj:=Workobject_1;
MoveL RelTool (p1,3.000000,12.500000,7.500000,\Rx:=0.000000,\Ry:=0.000000),vel1,zoneval,Extruder\WObj:=Workobject_1;
MoveL RelTool (p1,5.000000,13.000000,7.500000,\Rx:=0.000000,\Ry:=-0.000000),vel1,zoneval,Extruder\WObj:=Workobject_1;
MoveL RelTool (p1,7.500000,13.000000,7.500000,\Rx:=0.000000,\Ry:=-0.000000),vel1,zoneval,Extruder\WObj:=Workobject_1;
MoveL RelTool (p1,10.000000,13.000000,7.500000,\Rx:=0.000000,\Ry:=-0.000000),vel1,zoneval,Extruder\WObj:=Workobject_1;
MoveL RelTool (p1,12.500000,13.000000,7.500000,\Rx:=0.000000,\Ry:=-0.000000),vel1,zoneval,Extruder\WObj:=Workobject_1;
MoveL RelTool (p1,15.000000,13.000000,7.500000,\Rx:=0.000000,\Ry:=-0.000000),vel1,zoneval,Extruder\WObj:=Workobject_1;
MoveL RelTool (p1,17.500000,13.000000,7.549338,\Rx:=0.000000,\Ry:=-2.952187),vel1,zoneval,Extruder\WObj:=Workobject_1;
MoveL RelTool (p1,20.000000,13.000000,9.005299,\Rx:=0.000000,\Ry:=-11.722654),vel1,zoneval,Extruder\WObj:=Workobject_1;
MoveL RelTool (p1,22.500000,13.000000,11.676189,\Rx:=0.000000,\Ry:=-8.329854),vel1,zoneval,Extruder\WObj:=Workobject_1;
MoveL RelTool (p1,25.000000,13.000000,13.363865,\Rx:=0.000000,\Ry:=-6.543126),vel1,zoneval,Extruder\WObj:=Workobject_1;
MoveL RelTool (p1,27.500000,13.000000,14.596952,\Rx:=0.000000,\Ry:=-5.169413),vel1,zoneval,Extruder\WObj:=Workobject_1;
MoveL RelTool (p1,30.000000,13.000000,15.533723,\Rx:=0.000000,\Ry:=-4.264941),vel1,zoneval,Extruder\WObj:=Workobject_1;
MoveL RelTool (p1,32.500000,13.000000,16.262302,\Rx:=0.000000,\Ry:=-3.021941),vel1,zoneval,Extruder\WObj:=Workobject_1;
MoveL RelTool (p1,35.000000,13.000000,16.792830,\Rx:=0.000000,\Ry:=-2.385947),vel1,zoneval,Extruder\WObj:=Workobject_1;
MoveL RelTool (p1,37.500000,13.000000,17.166568,\Rx:=0.000000,\Ry:=-1.460854),vel1,zoneval,Extruder\WObj:=Workobject_1;
MoveL RelTool (p1,40.000000,13.000000,17.404149,\Rx:=0.000000,\Ry:=-0.649384),vel1,zoneval,Extruder\WObj:=Workobject_1;
MoveL RelTool (p1,42.500000,13.000000,17.492587,\Rx:=0.000000,\Ry:=0.009614),vel1,zoneval,Extruder\WObj:=Workobject_1;
MoveL RelTool (p1,45.000000,13.000000,17.446248,\Rx:=0.000000,\Ry:=0.497915),vel1,zoneval,Extruder\WObj:=Workobject_1;
MoveL RelTool (p1,47.500000,13.000000,17.267646,\Rx:=0.000000,\Ry:=1.437041),vel1,zoneval,Extruder\WObj:=Workobject_1;
MoveL RelTool (p1,50.000000,13.000000,16.932428,\Rx:=0.000000,\Ry:=1.939079),vel1,zoneval,Extruder\WObj:=Workobject_1;
MoveL RelTool (p1,52.500000,13.000000,16.460496,\Rx:=0.000000,\Ry:=2.957619),vel1,zoneval,Extruder\WObj:=Workobject_1;
MoveL RelTool (p1,55.000000,13.000000,15.795902,\Rx:=0.000000,\Ry:=3.558921),vel1,zoneval,Extruder\WObj:=Workobject_1;
MoveL RelTool (p1,57.500000,13.000000,14.937026,\Rx:=0.000000,\Ry:=4.724525),vel1,zoneval,Extruder\WObj:=Workobject_1;
MoveL RelTool (p1,60.000000,13.000000,13.809195,\Rx:=0.000000,\Ry:=5.980383),vel1,zoneval,Extruder\WObj:=Workobject_1;
MoveL RelTool (p1,62.500000,13.000000,12.303220,\Rx:=0.000000,\Ry:=8.147456),vel1,zoneval,Extruder\WObj:=Workobject_1;
MoveL RelTool (p1,65.000000,13.000000,10.062121,\Rx:=0.000000,\Ry:=11.495676),vel1,zoneval,Extruder\WObj:=Workobject_1;
MoveL RelTool (p1,67.500000,13.000000,7.780757,\Rx:=0.000000,\Ry:=3.821551),vel1,zoneval,Extruder\WObj:=Workobject_1;
MoveL RelTool (p1,70.000000,13.000000,7.500000,\Rx:=0.000000,\Ry:=-0.000000),vel1,zoneval,Extruder\WObj:=Workobject_1;
MoveL RelTool (p1,72.500000,13.000000,7.500000,\Rx:=0.000000,\Ry:=-0.000000),vel1,zoneval,Extruder\WObj:=Workobject_1;
MoveL RelTool (p1,75.000000,13.000000,7.500000,\Rx:=0.000000,\Ry:=-0.000000),vel1,zoneval,Extruder\WObj:=Workobject_1;
MoveL RelTool (p1,77.500000,13.000000,7.500000,\Rx:=0.000000,\Ry:=-0.000000),vel1,zoneval,Extruder\WObj:=Workobject_1;
MoveL RelTool (p1,80.000000,13.000000,7.500000,\Rx:=0.000000,\Ry:=-0.000000),vel1,zoneval,Extruder\WObj:=Workobject_1;
MoveL RelTool (p1,82.500000,13.000000,7.500000,\Rx:=0.000000,\Ry:=-0.000000),vel1,zoneval,Extruder\WObj:=Workobject_1;
MoveL RelTool (p1,80.500000,13.500000,7.500000,\Rx:=0.000000,\Ry:=0.000000),vel1,zoneval,Extruder\WObj:=Workobject_1;
MoveL RelTool (p1,78.000000,13.500000,7.500000,\Rx:=0.000000,\Ry:=0.000000),vel1,zoneval,Extruder\WObj:=Workobject_1;
MoveL RelTool (p1,75.500000,13.500000,7.500000,\Rx:=0.000000,\Ry:=0.000000),vel1,zoneval,Extruder\WObj:=Workobject_1;
MoveL RelTool (p1,73.000000,13.500000,7.500000,\Rx:=0.000000,\Ry:=0.000000),vel1,zoneval,Extruder\WObj:=Workobject_1;
MoveL RelTool (p1,70.500000,13.500000,7.500000,\Rx:=0.000000,\Ry:=0.000000),vel1,zoneval,Extruder\WObj:=Workobject_1;
MoveL RelTool (p1,68.000000,13.500000,7.626010,\Rx:=0.000000,\Ry:=3.821551),vel1,zoneval,Extruder\WObj:=Workobject_1;
MoveL RelTool (p1,65.500000,13.500000,9.428317,\Rx:=0.000000,\Ry:=11.492240),vel1,zoneval,Extruder\WObj:=Workobject_1;
MoveL RelTool (p1,63.000000,13.500000,11.932053,\Rx:=0.000000,\Ry:=8.135828),vel1,zoneval,Extruder\WObj:=Workobject_1;
MoveL RelTool (p1,60.500000,13.500000,13.555245,\Rx:=0.000000,\Ry:=5.992023),vel1,zoneval,Extruder\WObj:=Workobject_1;
MoveL RelTool (p1,58.000000,13.500000,14.743190,\Rx:=0.000000,\Ry:=4.720141),vel1,zoneval,Extruder\WObj:=Workobject_1;
MoveL RelTool (p1,55.500000,13.500000,15.653270,\Rx:=0.000000,\Ry:=3.576897),vel1,zoneval,Extruder\WObj:=Workobject_1;
MoveL RelTool (p1,53.000000,13.500000,16.342233,\Rx:=0.000000,\Ry:=2.980824),vel1,zoneval,Extruder\WObj:=Workobject_1;
MoveL RelTool (p1,50.500000,13.500000,16.856164,\Rx:=0.000000,\Ry:=1.948768),vel1,zoneval,Extruder\WObj:=Workobject_1;
MoveL RelTool (p1,48.000000,13.500000,17.210655,\Rx:=0.000000,\Ry:=1.465724),vel1,zoneval,Extruder\WObj:=Workobject_1;
MoveL RelTool (p1,45.500000,13.500000,17.426504,\Rx:=0.000000,\Ry:=0.497915),vel1,zoneval,Extruder\WObj:=Workobject_1;
MoveL RelTool (p1,43.000000,13.500000,17.492095,\Rx:=0.000000,\Ry:=0.009614),vel1,zoneval,Extruder\WObj:=Workobject_1;
MoveL RelTool (p1,40.500000,13.500000,17.430570,\Rx:=0.000000,\Ry:=-0.679887),vel1,zoneval,Extruder\WObj:=Workobject_1;
MoveL RelTool (p1,38.000000,13.500000,17.224829,\Rx:=0.000000,\Ry:=-1.460854),vel1,zoneval,Extruder\WObj:=Workobject_1;
MoveL RelTool (p1,35.500000,13.500000,16.887333,\Rx:=0.000000,\Ry:=-2.343245),vel1,zoneval,Extruder\WObj:=Workobject_1;
MoveL RelTool (p1,33.000000,13.500000,16.383138,\Rx:=0.000000,\Ry:=-3.021941),vel1,zoneval,Extruder\WObj:=Workobject_1;
MoveL RelTool (p1,30.500000,13.500000,15.708122,\Rx:=0.000000,\Ry:=-4.251753),vel1,zoneval,Extruder\WObj:=Workobject_1;
MoveL RelTool (p1,28.000000,13.500000,14.811558,\Rx:=0.000000,\Ry:=-5.142472),vel1,zoneval,Extruder\WObj:=Workobject_1;
MoveL RelTool (p1,25.500000,13.500000,13.645784,\Rx:=0.000000,\Ry:=-6.534244),vel1,zoneval,Extruder\WObj:=Workobject_1;
MoveL RelTool (p1,23.000000,13.500000,12.059406,\Rx:=0.000000,\Ry:=-8.317990),vel1,zoneval,Extruder\WObj:=Workobject_1;
MoveL RelTool (p1,20.500000,13.500000,9.662966,\Rx:=0.000000,\Ry:=-11.723467),vel1,zoneval,Extruder\WObj:=Workobject_1;
MoveL RelTool (p1,18.000000,13.500000,7.667393,\Rx:=0.000000,\Ry:=-2.952187),vel1,zoneval,Extruder\WObj:=Workobject_1;
MoveL RelTool (p1,15.500000,13.500000,7.500000,\Rx:=0.000000,\Ry:=0.000000),vel1,zoneval,Extruder\WObj:=Workobject_1;
MoveL RelTool (p1,13.000000,13.500000,7.500000,\Rx:=0.000000,\Ry:=0.000000),vel1,zoneval,Extruder\WObj:=Workobject_1;
MoveL RelTool (p1,10.500000,13.500000,7.500000,\Rx:=0.000000,\Ry:=0.000000),vel1,zoneval,Extruder\WObj:=Workobject_1;
MoveL RelTool (p1,8.000000,13.500000,7.500000,\Rx:=0.000000,\Ry:=0.000000),vel1,zoneval,Extruder\WObj:=Workobject_1;
MoveL RelTool (p1,5.500000,13.500000,7.500000,\Rx:=0.000000,\Ry:=0.000000),vel1,zoneval,Extruder\WObj:=Workobject_1;
MoveL RelTool (p1,3.000000,13.500000,7.500000,\Rx:=0.000000,\Ry:=0.000000),vel1,zoneval,Extruder\WObj:=Workobject_1;
MoveL RelTool (p1,5.000000,14.000000,7.500000,\Rx:=0.000000,\Ry:=-0.000000),vel1,zoneval,Extruder\WObj:=Workobject_1;
MoveL RelTool (p1,7.500000,14.000000,7.500000,\Rx:=0.000000,\Ry:=-0.000000),vel1,zoneval,Extruder\WObj:=Workobject_1;
MoveL RelTool (p1,10.000000,14.000000,7.500000,\Rx:=0.000000,\Ry:=-0.000000),vel1,zoneval,Extruder\WObj:=Workobject_1;
MoveL RelTool (p1,12.500000,14.000000,7.500000,\Rx:=0.000000,\Ry:=-0.000000),vel1,zoneval,Extruder\WObj:=Workobject_1;
MoveL RelTool (p1,15.000000,14.000000,7.500000,\Rx:=0.000000,\Ry:=-0.000000),vel1,zoneval,Extruder\WObj:=Workobject_1;
MoveL RelTool (p1,17.500000,14.000000,7.549338,\Rx:=0.000000,\Ry:=-2.952187),vel1,zoneval,Extruder\WObj:=Workobject_1;
MoveL RelTool (p1,20.000000,14.000000,9.005299,\Rx:=0.000000,\Ry:=-11.721669),vel1,zoneval,Extruder\WObj:=Workobject_1;
MoveL RelTool (p1,22.500000,14.000000,11.677209,\Rx:=0.000000,\Ry:=-8.306110),vel1,zoneval,Extruder\WObj:=Workobject_1;
MoveL RelTool (p1,25.000000,14.000000,13.364138,\Rx:=0.000000,\Ry:=-6.525355),vel1,zoneval,Extruder\WObj:=Workobject_1;
MoveL RelTool (p1,27.500000,14.000000,14.598779,\Rx:=0.000000,\Ry:=-5.115484),vel1,zoneval,Extruder\WObj:=Workobject_1;
